(* Logix 5000 project; controller LeakTestAuto vendor 1 type 14 code 226 rev 37.11; software revision 37.01; part 3 of 14 *)

        [3].Detailed.element_data[8].Variable_code := 59, [3].Detailed.element_data[8].prec_code := 2, [3].Detailed.element_data[8].Unit_code := 60, [3].Detailed.element_data[8].result_measurement := 1.0002404, [3].Detailed.element_data[9].Variable_code := 12, [3].Detailed.element_data[9].prec_code := 3, [3].Detailed.element_data[9].Unit_code := 12, [3].Detailed.element_data[9].result_measurement := 5.000001, [3].Detailed.element_data[10].Variable_code := 62, [3].Detailed.element_data[10].prec_code := 2, [3].Detailed.element_data[10].Unit_code := 60, [3].Detailed.element_data[10].result_measurement := 1.1002644, [3].Detailed.element_data[11].Variable_code := 21, [3].Detailed.element_data[11].prec_code := 3, [3].Detailed.element_data[11].Unit_code := 41, [3].Detailed.element_data[11].result_measurement := 0.0015180558, [3].Detailed.element_data[12].Variable_code := 25, [3].Detailed.element_data[12].prec_code := 3, [3].Detailed.element_data[12].Unit_code := 41, [3].Detailed.element_data[12].result_measurement := 0.021727756, [3].Detailed.element_data[13].Variable_code := 216, [3].Detailed.element_data[13].prec_code := 3, [3].Detailed.element_data[13].Unit_code := 41, [3].Detailed.element_data[13].result_measurement := 0.00085681677, [3].Detailed.element_data[14].Variable_code := 218, [3].Detailed.element_data[14].prec_code := 3, [3].Detailed.element_data[14].Unit_code := 41, [3].Detailed.element_data[14].result_measurement := 0.01094304, [3].Detailed.element_data[15].Variable_code := 295, [3].Detailed.element_data[15].prec_code := 3, [3].Detailed.element_data[15].Unit_code := 12, [3].Detailed.element_data[15].result_measurement := 5.1383443, [4].UID := 41965, [4].Basic.unique_id := 41965, [4].Basic.channel_num := 1, [4].Basic.program_num := 2, [4].Basic.evaluation_code := 1, [4].Basic.test_port := 1, [4].Basic.year := 26, [4].Basic.month := 6, [4].Basic.date := 4, [4].Basic.hour := 15, [4].Basic.minute := 7, [4].Basic.second := 53, [4].Basic.flags := 12, [4].Basic.Num_tests := 1, [4].Basic.test_elements.test_type := 66, [4].Basic.test_elements.test_eval := 1, [4].Basic.test_elements.num_elements := 16, [4].Detailed.unique_id := 41965, [4].Detailed.num_elements := 16, [4].Detailed.Test_Type := 66, [4].Detailed.element_data[0].Variable_code := 61, [4].Detailed.element_data[0].prec_code := 2, [4].Detailed.element_data[0].Unit_code := 60, [4].Detailed.element_data[0].result_measurement := -0.06593764, [4].Detailed.element_data[1].Variable_code := 28, [4].Detailed.element_data[1].prec_code := 3, [4].Detailed.element_data[1].Unit_code := 41, [4].Detailed.element_data[1].result_measurement := 0.00029802322,
        [4].Detailed.element_data[2].Variable_code := 13, [4].Detailed.element_data[2].prec_code := 3, [4].Detailed.element_data[2].Unit_code := 12, [4].Detailed.element_data[2].result_measurement := 5.1366444, [4].Detailed.element_data[3].Variable_code := 75, [4].Detailed.element_data[3].prec_code := 2, [4].Detailed.element_data[3].Unit_code := 60, [4].Detailed.element_data[4].Variable_code := 60, [4].Detailed.element_data[4].prec_code := 2, [4].Detailed.element_data[4].Unit_code := 60, [4].Detailed.element_data[4].result_measurement := -0.06984919, [4].Detailed.element_data[5].Variable_code := 56, [4].Detailed.element_data[5].prec_code := 3, [4].Detailed.element_data[5].Unit_code := 41, [4].Detailed.element_data[5].result_measurement := 0.00021420419, [4].Detailed.element_data[6].Variable_code := 55, [4].Detailed.element_data[6].prec_code := 3, [4].Detailed.element_data[6].Unit_code := 12, [4].Detailed.element_data[6].result_measurement := 5.1366444, [4].Detailed.element_data[7].Variable_code := 58, [4].Detailed.element_data[7].prec_code := 2, [4].Detailed.element_data[7].Unit_code := 60, [4].Detailed.element_data[7].result_measurement := -1.0002404, [4].Detailed.element_data[8].Variable_code := 59, [4].Detailed.element_data[8].prec_code := 2, [4].Detailed.element_data[8].Unit_code := 60, [4].Detailed.element_data[8].result_measurement := 1.0002404, [4].Detailed.element_data[9].Variable_code := 12, [4].Detailed.element_data[9].prec_code := 3, [4].Detailed.element_data[9].Unit_code := 12, [4].Detailed.element_data[9].result_measurement := 5.000001, [4].Detailed.element_data[10].Variable_code := 62, [4].Detailed.element_data[10].prec_code := 2, [4].Detailed.element_data[10].Unit_code := 60, [4].Detailed.element_data[10].result_measurement := 1.1002644, [4].Detailed.element_data[11].Variable_code := 21, [4].Detailed.element_data[11].prec_code := 3, [4].Detailed.element_data[11].Unit_code := 41, [4].Detailed.element_data[11].result_measurement := 0.0015180558, [4].Detailed.element_data[12].Variable_code := 25, [4].Detailed.element_data[12].prec_code := 3, [4].Detailed.element_data[12].Unit_code := 41, [4].Detailed.element_data[12].result_measurement := 0.021727756, [4].Detailed.element_data[13].Variable_code := 216, [4].Detailed.element_data[13].prec_code := 3, [4].Detailed.element_data[13].Unit_code := 41, [4].Detailed.element_data[13].result_measurement := 0.00085681677, [4].Detailed.element_data[14].Variable_code := 218, [4].Detailed.element_data[14].prec_code := 3, [4].Detailed.element_data[14].Unit_code := 41, [4].Detailed.element_data[14].result_measurement := 0.01094304, [4].Detailed.element_data[15].Variable_code := 295, [4].Detailed.element_data[15].prec_code := 3, [4].Detailed.element_data[15].Unit_code := 12, [4].Detailed.element_data[15].result_measurement := 5.138372, [5].UID := 41968, [5].Basic.unique_id := 41968, [5].Basic.channel_num := 1, [5].Basic.program_num := 2, [5].Basic.evaluation_code := 1,
        [5].Basic.test_port := 1, [5].Basic.year := 26, [5].Basic.month := 6, [5].Basic.date := 4, [5].Basic.hour := 15, [5].Basic.minute := 9, [5].Basic.second := 31, [5].Basic.flags := 12, [5].Basic.Num_tests := 1, [5].Basic.test_elements.test_type := 66, [5].Basic.test_elements.test_eval := 1, [5].Basic.test_elements.num_elements := 16, [5].Detailed.unique_id := 41968, [5].Detailed.num_elements := 16, [5].Detailed.Test_Type := 66, [5].Detailed.element_data[0].Variable_code := 61, [5].Detailed.element_data[0].prec_code := 2, [5].Detailed.element_data[0].Unit_code := 60, [5].Detailed.element_data[0].result_measurement := -0.054761767, [5].Detailed.element_data[1].Variable_code := 28, [5].Detailed.element_data[1].prec_code := 3, [5].Detailed.element_data[1].Unit_code := 41, [5].Detailed.element_data[1].result_measurement := 0.0005075708, [5].Detailed.element_data[2].Variable_code := 13, [5].Detailed.element_data[2].prec_code := 3, [5].Detailed.element_data[2].Unit_code := 12, [5].Detailed.element_data[2].result_measurement := 5.1372128, [5].Detailed.element_data[3].Variable_code := 75, [5].Detailed.element_data[3].prec_code := 2, [5].Detailed.element_data[3].Unit_code := 60, [5].Detailed.element_data[4].Variable_code := 60, [5].Detailed.element_data[4].prec_code := 2, [5].Detailed.element_data[4].Unit_code := 60, [5].Detailed.element_data[4].result_measurement := -0.05811453, [5].Detailed.element_data[5].Variable_code := 56, [5].Detailed.element_data[5].prec_code := 3, [5].Detailed.element_data[5].Unit_code := 41, [5].Detailed.element_data[5].result_measurement := 0.0003213063, [5].Detailed.element_data[6].Variable_code := 55, [5].Detailed.element_data[6].prec_code := 3, [5].Detailed.element_data[6].Unit_code := 12, [5].Detailed.element_data[6].result_measurement := 5.1372128, [5].Detailed.element_data[7].Variable_code := 58, [5].Detailed.element_data[7].prec_code := 2, [5].Detailed.element_data[7].Unit_code := 60, [5].Detailed.element_data[7].result_measurement := -1.0002404, [5].Detailed.element_data[8].Variable_code := 59, [5].Detailed.element_data[8].prec_code := 2, [5].Detailed.element_data[8].Unit_code := 60, [5].Detailed.element_data[8].result_measurement := 1.0002404, [5].Detailed.element_data[9].Variable_code := 12, [5].Detailed.element_data[9].prec_code := 3, [5].Detailed.element_data[9].Unit_code := 12, [5].Detailed.element_data[9].result_measurement := 5.000001, [5].Detailed.element_data[10].Variable_code := 62, [5].Detailed.element_data[10].prec_code := 2, [5].Detailed.element_data[10].Unit_code := 60, [5].Detailed.element_data[10].result_measurement := 1.1002644, [5].Detailed.element_data[11].Variable_code := 21, [5].Detailed.element_data[11].prec_code := 3,
        [5].Detailed.element_data[11].Unit_code := 41, [5].Detailed.element_data[11].result_measurement := 0.0015180558, [5].Detailed.element_data[12].Variable_code := 25, [5].Detailed.element_data[12].prec_code := 3, [5].Detailed.element_data[12].Unit_code := 41, [5].Detailed.element_data[12].result_measurement := 0.021727756, [5].Detailed.element_data[13].Variable_code := 216, [5].Detailed.element_data[13].prec_code := 3, [5].Detailed.element_data[13].Unit_code := 41, [5].Detailed.element_data[13].result_measurement := 0.00085681677, [5].Detailed.element_data[14].Variable_code := 218, [5].Detailed.element_data[14].prec_code := 3, [5].Detailed.element_data[14].Unit_code := 41, [5].Detailed.element_data[14].result_measurement := 0.01094304, [5].Detailed.element_data[15].Variable_code := 295, [5].Detailed.element_data[15].prec_code := 3, [5].Detailed.element_data[15].Unit_code := 12, [5].Detailed.element_data[15].result_measurement := 5.139271, [6].UID := 42010, [6].Basic.unique_id := 42010, [6].Basic.channel_num := 1, [6].Basic.program_num := 2, [6].Basic.evaluation_code := 1, [6].Basic.test_port := 1, [6].Basic.year := 26, [6].Basic.month := 6, [6].Basic.date := 5, [6].Basic.hour := 10, [6].Basic.minute := 13, [6].Basic.second := 42, [6].Basic.flags := 12, [6].Basic.Num_tests := 1, [6].Basic.test_elements.test_type := 66, [6].Basic.test_elements.test_eval := 1, [6].Basic.test_elements.num_elements := 16, [6].Detailed.unique_id := 42010, [6].Detailed.num_elements := 16, [6].Detailed.Test_Type := 66, [6].Detailed.element_data[0].Variable_code := 61, [6].Detailed.element_data[0].prec_code := 2, [6].Detailed.element_data[0].Unit_code := 60, [6].Detailed.element_data[0].result_measurement := -0.067055225, [6].Detailed.element_data[1].Variable_code := 28, [6].Detailed.element_data[1].prec_code := 3, [6].Detailed.element_data[1].Unit_code := 41, [6].Detailed.element_data[1].result_measurement := 0.00027939677, [6].Detailed.element_data[2].Variable_code := 13, [6].Detailed.element_data[2].prec_code := 3, [6].Detailed.element_data[2].Unit_code := 12, [6].Detailed.element_data[2].result_measurement := 5.1023254, [6].Detailed.element_data[3].Variable_code := 75, [6].Detailed.element_data[3].prec_code := 2, [6].Detailed.element_data[3].Unit_code := 60, [6].Detailed.element_data[4].Variable_code := 60, [6].Detailed.element_data[4].prec_code := 2, [6].Detailed.element_data[4].Unit_code := 60, [6].Detailed.element_data[4].result_measurement := -0.07208437, [6].Detailed.element_data[5].Variable_code := 56, [6].Detailed.element_data[5].prec_code := 3, [6].Detailed.element_data[5].Unit_code := 41,
        [6].Detailed.element_data[5].result_measurement := 0.00019092113, [6].Detailed.element_data[6].Variable_code := 55, [6].Detailed.element_data[6].prec_code := 3, [6].Detailed.element_data[6].Unit_code := 12, [6].Detailed.element_data[6].result_measurement := 5.1023254, [6].Detailed.element_data[7].Variable_code := 58, [6].Detailed.element_data[7].prec_code := 2, [6].Detailed.element_data[7].Unit_code := 60, [6].Detailed.element_data[7].result_measurement := -1.0002404, [6].Detailed.element_data[8].Variable_code := 59, [6].Detailed.element_data[8].prec_code := 2, [6].Detailed.element_data[8].Unit_code := 60, [6].Detailed.element_data[8].result_measurement := 1.0002404, [6].Detailed.element_data[9].Variable_code := 12, [6].Detailed.element_data[9].prec_code := 3, [6].Detailed.element_data[9].Unit_code := 12, [6].Detailed.element_data[9].result_measurement := 5.000001, [6].Detailed.element_data[10].Variable_code := 62, [6].Detailed.element_data[10].prec_code := 2, [6].Detailed.element_data[10].Unit_code := 60, [6].Detailed.element_data[10].result_measurement := 1.1002644, [6].Detailed.element_data[11].Variable_code := 21, [6].Detailed.element_data[11].prec_code := 3, [6].Detailed.element_data[11].Unit_code := 41, [6].Detailed.element_data[11].result_measurement := 0.0015180558, [6].Detailed.element_data[12].Variable_code := 25, [6].Detailed.element_data[12].prec_code := 3, [6].Detailed.element_data[12].Unit_code := 41, [6].Detailed.element_data[12].result_measurement := 0.021727756, [6].Detailed.element_data[13].Variable_code := 216, [6].Detailed.element_data[13].prec_code := 3, [6].Detailed.element_data[13].Unit_code := 41, [6].Detailed.element_data[13].result_measurement := 0.00085681677, [6].Detailed.element_data[14].Variable_code := 218, [6].Detailed.element_data[14].prec_code := 3, [6].Detailed.element_data[14].Unit_code := 41, [6].Detailed.element_data[14].result_measurement := 0.01094304, [6].Detailed.element_data[15].Variable_code := 295, [6].Detailed.element_data[15].prec_code := 3, [6].Detailed.element_data[15].Unit_code := 12, [6].Detailed.element_data[15].result_measurement := 5.1039925, [7].UID := 42013, [7].Basic.unique_id := 42013, [7].Basic.channel_num := 1, [7].Basic.program_num := 2, [7].Basic.evaluation_code := 1, [7].Basic.test_port := 1, [7].Basic.year := 26, [7].Basic.month := 6, [7].Basic.date := 5, [7].Basic.hour := 10, [7].Basic.minute := 17, [7].Basic.second := 34, [7].Basic.flags := 12, [7].Basic.Num_tests := 1, [7].Basic.test_elements.test_type := 66, [7].Basic.test_elements.test_eval := 1, [7].Basic.test_elements.num_elements := 16, [7].Detailed.unique_id := 42013, [7].Detailed.num_elements := 16,
        [7].Detailed.Test_Type := 66, [7].Detailed.element_data[0].Variable_code := 61, [7].Detailed.element_data[0].prec_code := 2, [7].Detailed.element_data[0].Unit_code := 60, [7].Detailed.element_data[0].result_measurement := -0.07040799, [7].Detailed.element_data[1].Variable_code := 28, [7].Detailed.element_data[1].prec_code := 3, [7].Detailed.element_data[1].Unit_code := 41, [7].Detailed.element_data[1].result_measurement := 0.00022351742, [7].Detailed.element_data[2].Variable_code := 13, [7].Detailed.element_data[2].prec_code := 3, [7].Detailed.element_data[2].Unit_code := 12, [7].Detailed.element_data[2].result_measurement := 5.101585, [7].Detailed.element_data[3].Variable_code := 75, [7].Detailed.element_data[3].prec_code := 2, [7].Detailed.element_data[3].Unit_code := 60, [7].Detailed.element_data[4].Variable_code := 60, [7].Detailed.element_data[4].prec_code := 2, [7].Detailed.element_data[4].Unit_code := 60, [7].Detailed.element_data[4].result_measurement := -0.07711351, [7].Detailed.element_data[5].Variable_code := 56, [7].Detailed.element_data[5].prec_code := 3, [7].Detailed.element_data[5].Unit_code := 41, [7].Detailed.element_data[5].result_measurement := 0.00014901161, [7].Detailed.element_data[6].Variable_code := 55, [7].Detailed.element_data[6].prec_code := 3, [7].Detailed.element_data[6].Unit_code := 12, [7].Detailed.element_data[6].result_measurement := 5.101585, [7].Detailed.element_data[7].Variable_code := 58, [7].Detailed.element_data[7].prec_code := 2, [7].Detailed.element_data[7].Unit_code := 60, [7].Detailed.element_data[7].result_measurement := -1.0002404, [7].Detailed.element_data[8].Variable_code := 59, [7].Detailed.element_data[8].prec_code := 2, [7].Detailed.element_data[8].Unit_code := 60, [7].Detailed.element_data[8].result_measurement := 1.0002404, [7].Detailed.element_data[9].Variable_code := 12, [7].Detailed.element_data[9].prec_code := 3, [7].Detailed.element_data[9].Unit_code := 12, [7].Detailed.element_data[9].result_measurement := 5.000001, [7].Detailed.element_data[10].Variable_code := 62, [7].Detailed.element_data[10].prec_code := 2, [7].Detailed.element_data[10].Unit_code := 60, [7].Detailed.element_data[10].result_measurement := 1.1002644, [7].Detailed.element_data[11].Variable_code := 21, [7].Detailed.element_data[11].prec_code := 3, [7].Detailed.element_data[11].Unit_code := 41, [7].Detailed.element_data[11].result_measurement := 0.0015180558, [7].Detailed.element_data[12].Variable_code := 25, [7].Detailed.element_data[12].prec_code := 3, [7].Detailed.element_data[12].Unit_code := 41, [7].Detailed.element_data[12].result_measurement := 0.021727756, [7].Detailed.element_data[13].Variable_code := 216, [7].Detailed.element_data[13].prec_code := 3, [7].Detailed.element_data[13].Unit_code := 41, [7].Detailed.element_data[13].result_measurement := 0.00085681677, [7].Detailed.element_data[14].Variable_code := 218, [7].Detailed.element_data[14].prec_code := 3, [7].Detailed.element_data[14].Unit_code := 41, [7].Detailed.element_data[14].result_measurement := 0.01094304,
        [7].Detailed.element_data[15].Variable_code := 295, [7].Detailed.element_data[15].prec_code := 3, [7].Detailed.element_data[15].Unit_code := 12, [7].Detailed.element_data[15].result_measurement := 5.103038, [8].UID := 42016, [8].Basic.unique_id := 42016, [8].Basic.channel_num := 1, [8].Basic.program_num := 2, [8].Basic.evaluation_code := 1, [8].Basic.test_port := 1, [8].Basic.year := 26, [8].Basic.month := 6, [8].Basic.date := 5, [8].Basic.hour := 10, [8].Basic.minute := 18, [8].Basic.second := 33, [8].Basic.flags := 12, [8].Basic.Num_tests := 1, [8].Basic.test_elements.test_type := 66, [8].Basic.test_elements.test_eval := 1, [8].Basic.test_elements.num_elements := 16, [8].Detailed.unique_id := 42016, [8].Detailed.num_elements := 16, [8].Detailed.Test_Type := 66, [8].Detailed.element_data[0].Variable_code := 61, [8].Detailed.element_data[0].prec_code := 2, [8].Detailed.element_data[0].Unit_code := 60, [8].Detailed.element_data[0].result_measurement := -0.0692904, [8].Detailed.element_data[1].Variable_code := 28, [8].Detailed.element_data[1].prec_code := 3, [8].Detailed.element_data[1].Unit_code := 41, [8].Detailed.element_data[1].result_measurement := 0.00023748726, [8].Detailed.element_data[2].Variable_code := 13, [8].Detailed.element_data[2].prec_code := 3, [8].Detailed.element_data[2].Unit_code := 12, [8].Detailed.element_data[2].result_measurement := 5.1036057, [8].Detailed.element_data[3].Variable_code := 75, [8].Detailed.element_data[3].prec_code := 2, [8].Detailed.element_data[3].Unit_code := 60, [8].Detailed.element_data[4].Variable_code := 60, [8].Detailed.element_data[4].prec_code := 2, [8].Detailed.element_data[4].Unit_code := 60, [8].Detailed.element_data[4].result_measurement := -0.073201954, [8].Detailed.element_data[5].Variable_code := 56, [8].Detailed.element_data[5].prec_code := 3, [8].Detailed.element_data[5].Unit_code := 41, [8].Detailed.element_data[5].result_measurement := 0.0001816079, [8].Detailed.element_data[6].Variable_code := 55, [8].Detailed.element_data[6].prec_code := 3, [8].Detailed.element_data[6].Unit_code := 12, [8].Detailed.element_data[6].result_measurement := 5.1036057, [8].Detailed.element_data[7].Variable_code := 58, [8].Detailed.element_data[7].prec_code := 2, [8].Detailed.element_data[7].Unit_code := 60, [8].Detailed.element_data[7].result_measurement := -1.0002404, [8].Detailed.element_data[8].Variable_code := 59, [8].Detailed.element_data[8].prec_code := 2, [8].Detailed.element_data[8].Unit_code := 60, [8].Detailed.element_data[8].result_measurement := 1.0002404, [8].Detailed.element_data[9].Variable_code := 12,
        [8].Detailed.element_data[9].prec_code := 3, [8].Detailed.element_data[9].Unit_code := 12, [8].Detailed.element_data[9].result_measurement := 5.000001, [8].Detailed.element_data[10].Variable_code := 62, [8].Detailed.element_data[10].prec_code := 2, [8].Detailed.element_data[10].Unit_code := 60, [8].Detailed.element_data[10].result_measurement := 1.1002644, [8].Detailed.element_data[11].Variable_code := 21, [8].Detailed.element_data[11].prec_code := 3, [8].Detailed.element_data[11].Unit_code := 41, [8].Detailed.element_data[11].result_measurement := 0.0015180558, [8].Detailed.element_data[12].Variable_code := 25, [8].Detailed.element_data[12].prec_code := 3, [8].Detailed.element_data[12].Unit_code := 41, [8].Detailed.element_data[12].result_measurement := 0.021727756, [8].Detailed.element_data[13].Variable_code := 216, [8].Detailed.element_data[13].prec_code := 3, [8].Detailed.element_data[13].Unit_code := 41, [8].Detailed.element_data[13].result_measurement := 0.00085681677, [8].Detailed.element_data[14].Variable_code := 218, [8].Detailed.element_data[14].prec_code := 3, [8].Detailed.element_data[14].Unit_code := 41, [8].Detailed.element_data[14].result_measurement := 0.01094304, [8].Detailed.element_data[15].Variable_code := 295, [8].Detailed.element_data[15].prec_code := 3, [8].Detailed.element_data[15].Unit_code := 12, [8].Detailed.element_data[15].result_measurement := 5.1049933);
   CTS2_ResultHistoryVol : udt_CTS_RESULT[10] := ([0].UID := 41958, [0].Basic.unique_id := 41958, [0].Basic.channel_num := 1, [0].Basic.program_num := 1, [0].Basic.evaluation_code := 1, [0].Basic.test_port := 1, [0].Basic.year := 26, [0].Basic.month := 6, [0].Basic.date := 4, [0].Basic.hour := 15, [0].Basic.minute := 3, [0].Basic.second := 10, [0].Basic.flags := 12, [0].Basic.Num_tests := 1, [0].Basic.test_elements.test_type := 69, [0].Basic.test_elements.test_eval := 1, [0].Basic.test_elements.num_elements := 4, [0].Detailed.unique_id := 41958, [0].Detailed.num_elements := 4, [0].Detailed.Test_Type := 69, [0].Detailed.element_data[0].Variable_code := 245, [0].Detailed.element_data[0].prec_code := 2, [0].Detailed.element_data[0].Unit_code := 165, [0].Detailed.element_data[0].result_measurement := 186.90665, [0].Detailed.element_data[1].Variable_code := 13, [0].Detailed.element_data[1].prec_code := 3, [0].Detailed.element_data[1].Unit_code := 12, [0].Detailed.element_data[1].result_measurement := 1.7801206, [0].Detailed.element_data[2].Variable_code := 247, [0].Detailed.element_data[2].prec_code := 3, [0].Detailed.element_data[2].Unit_code := 12, [0].Detailed.element_data[2].result_measurement := 5.1072845, [0].Detailed.element_data[3].Variable_code := 295, [0].Detailed.element_data[3].prec_code := 3, [0].Detailed.element_data[3].Unit_code := 12, [0].Detailed.element_data[3].result_measurement := 5.1086583, [1].UID := 41961, [1].Basic.unique_id := 41961, [1].Basic.channel_num := 1, [1].Basic.program_num := 1, [1].Basic.evaluation_code := 1, [1].Basic.test_port := 1, [1].Basic.year := 26, [1].Basic.month := 6, [1].Basic.date := 4, [1].Basic.hour := 15, [1].Basic.minute := 6, [1].Basic.second := 33, [1].Basic.flags := 12, [1].Basic.Num_tests := 1, [1].Basic.test_elements.test_type := 69, [1].Basic.test_elements.test_eval := 1, [1].Basic.test_elements.num_elements := 4, [1].Detailed.unique_id := 41961, [1].Detailed.num_elements := 4, [1].Detailed.Test_Type := 69, [1].Detailed.element_data[0].Variable_code := 245, [1].Detailed.element_data[0].prec_code := 2, [1].Detailed.element_data[0].Unit_code := 165, [1].Detailed.element_data[0].result_measurement := 186.6259,
        [1].Detailed.element_data[1].Variable_code := 13, [1].Detailed.element_data[1].prec_code := 3, [1].Detailed.element_data[1].Unit_code := 12, [1].Detailed.element_data[1].result_measurement := 1.7820624, [1].Detailed.element_data[2].Variable_code := 247, [1].Detailed.element_data[2].prec_code := 3, [1].Detailed.element_data[2].Unit_code := 12, [1].Detailed.element_data[2].result_measurement := 5.1078525, [1].Detailed.element_data[3].Variable_code := 295, [1].Detailed.element_data[3].prec_code := 3, [1].Detailed.element_data[3].Unit_code := 12, [1].Detailed.element_data[3].result_measurement := 5.1083417, [2].UID := 41964, [2].Basic.unique_id := 41964, [2].Basic.channel_num := 1, [2].Basic.program_num := 1, [2].Basic.evaluation_code := 1, [2].Basic.test_port := 1, [2].Basic.year := 26, [2].Basic.month := 6, [2].Basic.date := 4, [2].Basic.hour := 15, [2].Basic.minute := 7, [2].Basic.second := 46, [2].Basic.flags := 12, [2].Basic.Num_tests := 1, [2].Basic.test_elements.test_type := 69, [2].Basic.test_elements.test_eval := 1, [2].Basic.test_elements.num_elements := 4, [2].Detailed.unique_id := 41964, [2].Detailed.num_elements := 4, [2].Detailed.Test_Type := 69, [2].Detailed.element_data[0].Variable_code := 245, [2].Detailed.element_data[0].prec_code := 2, [2].Detailed.element_data[0].Unit_code := 165, [2].Detailed.element_data[0].result_measurement := 186.70047, [2].Detailed.element_data[1].Variable_code := 13, [2].Detailed.element_data[1].prec_code := 3, [2].Detailed.element_data[1].Unit_code := 12, [2].Detailed.element_data[1].result_measurement := 1.7814804, [2].Detailed.element_data[2].Variable_code := 247, [2].Detailed.element_data[2].prec_code := 3, [2].Detailed.element_data[2].Unit_code := 12, [2].Detailed.element_data[2].result_measurement := 5.1075125, [2].Detailed.element_data[3].Variable_code := 295, [2].Detailed.element_data[3].prec_code := 3, [2].Detailed.element_data[3].Unit_code := 12, [2].Detailed.element_data[3].result_measurement := 5.1079783, [3].UID := 41967, [3].Basic.unique_id := 41967, [3].Basic.channel_num := 1, [3].Basic.program_num := 1, [3].Basic.evaluation_code := 1, [3].Basic.test_port := 1, [3].Basic.year := 26, [3].Basic.month := 6, [3].Basic.date := 4, [3].Basic.hour := 15, [3].Basic.minute := 9, [3].Basic.second := 24,
        [3].Basic.flags := 12, [3].Basic.Num_tests := 1, [3].Basic.test_elements.test_type := 69, [3].Basic.test_elements.test_eval := 1, [3].Basic.test_elements.num_elements := 4, [3].Detailed.unique_id := 41967, [3].Detailed.num_elements := 4, [3].Detailed.Test_Type := 69, [3].Detailed.element_data[0].Variable_code := 245, [3].Detailed.element_data[0].prec_code := 2, [3].Detailed.element_data[0].Unit_code := 165, [3].Detailed.element_data[0].result_measurement := 186.79054, [3].Detailed.element_data[1].Variable_code := 13, [3].Detailed.element_data[1].prec_code := 3, [3].Detailed.element_data[1].Unit_code := 12, [3].Detailed.element_data[1].result_measurement := 1.7802324, [3].Detailed.element_data[2].Variable_code := 247, [3].Detailed.element_data[2].prec_code := 3, [3].Detailed.element_data[2].Unit_code := 12, [3].Detailed.element_data[2].result_measurement := 5.1055384, [3].Detailed.element_data[3].Variable_code := 295, [3].Detailed.element_data[3].prec_code := 3, [3].Detailed.element_data[3].Unit_code := 12, [3].Detailed.element_data[3].result_measurement := 5.1066375, [4].UID := 42009, [4].Basic.unique_id := 42009, [4].Basic.channel_num := 1, [4].Basic.program_num := 1, [4].Basic.evaluation_code := 1, [4].Basic.test_port := 1, [4].Basic.year := 26, [4].Basic.month := 6, [4].Basic.date := 5, [4].Basic.hour := 10, [4].Basic.minute := 13, [4].Basic.second := 35, [4].Basic.flags := 12, [4].Basic.Num_tests := 1, [4].Basic.test_elements.test_type := 69, [4].Basic.test_elements.test_eval := 1, [4].Basic.test_elements.num_elements := 4, [4].Detailed.unique_id := 42009, [4].Detailed.num_elements := 4, [4].Detailed.Test_Type := 69, [4].Detailed.element_data[0].Variable_code := 245, [4].Detailed.element_data[0].prec_code := 2, [4].Detailed.element_data[0].Unit_code := 165, [4].Detailed.element_data[0].result_measurement := 185.74803, [4].Detailed.element_data[1].Variable_code := 13, [4].Detailed.element_data[1].prec_code := 3, [4].Detailed.element_data[1].Unit_code := 12, [4].Detailed.element_data[1].result_measurement := 1.7781556, [4].Detailed.element_data[2].Variable_code := 247, [4].Detailed.element_data[2].prec_code := 3, [4].Detailed.element_data[2].Unit_code := 12, [4].Detailed.element_data[2].result_measurement := 5.0810447, [4].Detailed.element_data[3].Variable_code := 295, [4].Detailed.element_data[3].prec_code := 3, [4].Detailed.element_data[3].Unit_code := 12, [4].Detailed.element_data[3].result_measurement := 5.081105,
        [5].UID := 42012, [5].Basic.unique_id := 42012, [5].Basic.channel_num := 1, [5].Basic.program_num := 1, [5].Basic.evaluation_code := 1, [5].Basic.test_port := 1, [5].Basic.year := 26, [5].Basic.month := 6, [5].Basic.date := 5, [5].Basic.hour := 10, [5].Basic.minute := 17, [5].Basic.second := 27, [5].Basic.flags := 12, [5].Basic.Num_tests := 1, [5].Basic.test_elements.test_type := 69, [5].Basic.test_elements.test_eval := 1, [5].Basic.test_elements.num_elements := 4, [5].Detailed.unique_id := 42012, [5].Detailed.num_elements := 4, [5].Detailed.Test_Type := 69, [5].Detailed.element_data[0].Variable_code := 245, [5].Detailed.element_data[0].prec_code := 2, [5].Detailed.element_data[0].Unit_code := 165, [5].Detailed.element_data[0].result_measurement := 185.72876, [5].Detailed.element_data[1].Variable_code := 13, [5].Detailed.element_data[1].prec_code := 3, [5].Detailed.element_data[1].Unit_code := 12, [5].Detailed.element_data[1].result_measurement := 1.7785281, [5].Detailed.element_data[2].Variable_code := 247, [5].Detailed.element_data[2].prec_code := 3, [5].Detailed.element_data[2].Unit_code := 12, [5].Detailed.element_data[2].result_measurement := 5.081766, [5].Detailed.element_data[3].Variable_code := 295, [5].Detailed.element_data[3].prec_code := 3, [5].Detailed.element_data[3].Unit_code := 12, [5].Detailed.element_data[3].result_measurement := 5.0830374, [6].UID := 42015, [6].Basic.unique_id := 42015, [6].Basic.channel_num := 1, [6].Basic.program_num := 1, [6].Basic.evaluation_code := 1, [6].Basic.test_port := 1, [6].Basic.year := 26, [6].Basic.month := 6, [6].Basic.date := 5, [6].Basic.hour := 10, [6].Basic.minute := 18, [6].Basic.second := 26, [6].Basic.flags := 12, [6].Basic.Num_tests := 1, [6].Basic.test_elements.test_type := 69, [6].Basic.test_elements.test_eval := 1, [6].Basic.test_elements.num_elements := 4, [6].Detailed.unique_id := 42015, [6].Detailed.num_elements := 4, [6].Detailed.Test_Type := 69, [6].Detailed.element_data[0].Variable_code := 245, [6].Detailed.element_data[0].prec_code := 2, [6].Detailed.element_data[0].Unit_code := 165, [6].Detailed.element_data[0].result_measurement := 185.95625,
        [6].Detailed.element_data[1].Variable_code := 13, [6].Detailed.element_data[1].prec_code := 3, [6].Detailed.element_data[1].Unit_code := 12, [6].Detailed.element_data[1].result_measurement := 1.778258, [6].Detailed.element_data[2].Variable_code := 247, [6].Detailed.element_data[2].prec_code := 3, [6].Detailed.element_data[2].Unit_code := 12, [6].Detailed.element_data[2].result_measurement := 5.08504, [6].Detailed.element_data[3].Variable_code := 295, [6].Detailed.element_data[3].prec_code := 3, [6].Detailed.element_data[3].Unit_code := 12, [6].Detailed.element_data[3].result_measurement := 5.086218, [7].UID := 42018, [7].Basic.unique_id := 42018, [7].Basic.channel_num := 1, [7].Basic.program_num := 1, [7].Basic.evaluation_code := 2, [7].Basic.test_port := 1, [7].Basic.year := 26, [7].Basic.month := 6, [7].Basic.date := 5, [7].Basic.hour := 10, [7].Basic.minute := 54, [7].Basic.second := 14, [7].Basic.flags := 12, [7].Basic.Num_tests := 1, [7].Basic.test_elements.test_type := 69, [7].Basic.test_elements.test_eval := 2, [7].Basic.test_elements.num_elements := 4, [7].Detailed.unique_id := 42018, [7].Detailed.num_elements := 4, [7].Detailed.Test_Type := 69, [7].Detailed.element_data[0].Variable_code := 245, [7].Detailed.element_data[0].prec_code := 2, [7].Detailed.element_data[0].Unit_code := 165, [7].Detailed.element_data[0].result_measurement := 1000.0, [7].Detailed.element_data[1].Variable_code := 13, [7].Detailed.element_data[1].prec_code := 3, [7].Detailed.element_data[1].Unit_code := 12, [7].Detailed.element_data[1].result_measurement := 0.0002933666, [7].Detailed.element_data[2].Variable_code := 247, [7].Detailed.element_data[2].prec_code := 3, [7].Detailed.element_data[2].Unit_code := 12, [7].Detailed.element_data[2].result_measurement := 5.0650864, [7].Detailed.element_data[3].Variable_code := 295, [7].Detailed.element_data[3].prec_code := 3, [7].Detailed.element_data[3].Unit_code := 12, [7].Detailed.element_data[3].result_measurement := 5.0667486, [8].UID := 42020, [8].Basic.unique_id := 42020, [8].Basic.channel_num := 1, [8].Basic.program_num := 1, [8].Basic.evaluation_code := 1, [8].Basic.test_port := 1, [8].Basic.year := 26, [8].Basic.month := 6, [8].Basic.date := 5, [8].Basic.hour := 10, [8].Basic.minute := 54, [8].Basic.second := 35,
        [8].Basic.flags := 12, [8].Basic.Num_tests := 1, [8].Basic.test_elements.test_type := 69, [8].Basic.test_elements.test_eval := 1, [8].Basic.test_elements.num_elements := 4, [8].Detailed.unique_id := 42020, [8].Detailed.num_elements := 4, [8].Detailed.Test_Type := 69, [8].Detailed.element_data[0].Variable_code := 245, [8].Detailed.element_data[0].prec_code := 2, [8].Detailed.element_data[0].Unit_code := 165, [8].Detailed.element_data[0].result_measurement := 186.5566, [8].Detailed.element_data[1].Variable_code := 13, [8].Detailed.element_data[1].prec_code := 3, [8].Detailed.element_data[1].Unit_code := 12, [8].Detailed.element_data[1].result_measurement := 1.768372, [8].Detailed.element_data[2].Variable_code := 247, [8].Detailed.element_data[2].prec_code := 3, [8].Detailed.element_data[2].Unit_code := 12, [8].Detailed.element_data[2].result_measurement := 5.0673866, [8].Detailed.element_data[3].Variable_code := 295, [8].Detailed.element_data[3].prec_code := 3, [8].Detailed.element_data[3].Unit_code := 12, [8].Detailed.element_data[3].result_measurement := 5.068574, [9].UID := 42023, [9].Basic.unique_id := 42023, [9].Basic.channel_num := 1, [9].Basic.program_num := 1, [9].Basic.evaluation_code := 1, [9].Basic.test_port := 1, [9].Basic.year := 26, [9].Basic.month := 6, [9].Basic.date := 5, [9].Basic.hour := 10, [9].Basic.minute := 55, [9].Basic.second := 43, [9].Basic.flags := 12, [9].Basic.Num_tests := 1, [9].Basic.test_elements.test_type := 69, [9].Basic.test_elements.test_eval := 1, [9].Basic.test_elements.num_elements := 4, [9].Detailed.unique_id := 42023, [9].Detailed.num_elements := 4, [9].Detailed.Test_Type := 69, [9].Detailed.element_data[0].Variable_code := 245, [9].Detailed.element_data[0].prec_code := 2, [9].Detailed.element_data[0].Unit_code := 165, [9].Detailed.element_data[0].result_measurement := 186.64526, [9].Detailed.element_data[1].Variable_code := 13, [9].Detailed.element_data[1].prec_code := 3, [9].Detailed.element_data[1].Unit_code := 12, [9].Detailed.element_data[1].result_measurement := 1.7689215, [9].Detailed.element_data[2].Variable_code := 247, [9].Detailed.element_data[2].prec_code := 3, [9].Detailed.element_data[2].Unit_code := 12, [9].Detailed.element_data[2].result_measurement := 5.07053, [9].Detailed.element_data[3].Variable_code := 295, [9].Detailed.element_data[3].prec_code := 3, [9].Detailed.element_data[3].Unit_code := 12, [9].Detailed.element_data[3].result_measurement := 5.0715685);
   CTS2_Seq : udt_SequenceStructure_X64 := (CycleDone := 1, CurrentStep := 9000, NextStep := 9000, ONS := -32767, StepHistory[0] := 1000, StepHistory[1] := 1010, StepHistory[2] := 1020, StepHistory[3] := 1030, StepHistory[4] := 2000, StepHistory[5] := 2010, StepHistory[6] := 2020, StepHistory[7] := 2030, StepHistory[8] := 2000, StepHistory[9] := 2010, StepHistory[10] := 2020, StepHistory[11] := 2030, StepHistory[12] := 9000, StepHistory[13] := 1000, StepHistory[14] := 1010, StepHistory[15] := 1020, StepHistory[16] := 1030, StepHistory[17] := 2000, StepHistory[18] := 2010, StepHistory[19] := 2020, StepHistory[20] := 2030, StepHistory[21] := 2000, StepHistory[22] := 2010, StepHistory[23] := 2020, StepHistory[24] := 2030, StepHistory[25] := 9000, StepHistory[26] := 1000, StepHistory[27] := 1010, StepHistory[28] := 1020, StepHistory[29] := 1030, StepHistory[30] := 2000, StepHistory[31] := 2010, StepHistory[32] := 2020, StepHistory[33] := 2030, StepHistory[34] := 9000, StepHistory[35] := 1000, StepHistory[36] := 1010, StepHistory[37] := 1020, StepHistory[38] := 1030, StepHistory[39] := 2000, StepHistory[40] := 2010, StepHistory[41] := 2020, StepHistory[42] := 2030, StepHistory[43] := 2000, StepHistory[44] := 2010, StepHistory[45] := 2020, StepHistory[46] := 2030, StepHistory[47] := 9000, StepHistory[48] := 1000, StepHistory[49] := 1010, StepHistory[50] := 1020, StepHistory[51] := 1030, StepHistory[52] := 2000, StepHistory[53] := 2010, StepHistory[54] := 2020, StepHistory[55] := 2030,
        StepHistory[56] := 2000, StepHistory[57] := 2010, StepHistory[58] := 2020, StepHistory[59] := 2030, StepHistory[60] := 9000, StepHistory[61] := 1000, StepHistory[62] := 1010, StepHistory[63] := 1020, AverageCycleTime := 1.0542, CycleTimeHistory[0] := 2.209, CycleTimeHistory[1] := 2.209, CycleTimeHistory[3] := 1.206, CycleTimeHistory[4] := 2.209, CycleTimeHistory[5] := 2.209, CycleTimeHistory[8] := 0.5, StepTimeHistory[1] := 0.199, StepTimeHistory[2] := 0.199, StepTimeHistory[3] := 0.199, StepTimeHistory[5] := 1.0, StepTimeHistory[6] := 1.0, StepTimeHistory[7] := 1.0, StepTimeHistory[9] := 0.999, StepTimeHistory[10] := 0.999, StepTimeHistory[11] := 0.999, StepTimeHistory[12] := 0.999, StepTimeHistory[14] := 0.199, StepTimeHistory[15] := 0.199, StepTimeHistory[16] := 0.199, StepTimeHistory[18] := 1.0, StepTimeHistory[19] := 1.0, StepTimeHistory[20] := 1.0, StepTimeHistory[22] := 0.999, StepTimeHistory[23] := 0.999, StepTimeHistory[24] := 0.999, StepTimeHistory[27] := 0.199, StepTimeHistory[28] := 0.199, StepTimeHistory[29] := 0.199, StepTimeHistory[31] := 1.0, StepTimeHistory[32] := 1.0, StepTimeHistory[33] := 1.0, StepTimeHistory[34] := 1.0, StepTimeHistory[36] := 0.199, StepTimeHistory[37] := 0.199, StepTimeHistory[38] := 0.199, StepTimeHistory[40] := 0.999, StepTimeHistory[41] := 0.999, StepTimeHistory[42] := 0.999, StepTimeHistory[44] := 1.0, StepTimeHistory[45] := 1.0, StepTimeHistory[46] := 1.0, StepTimeHistory[47] := 1.0, StepTimeHistory[49] := 0.2, StepTimeHistory[50] := 0.2, StepTimeHistory[51] := 0.2, StepTimeHistory[53] := 0.999, StepTimeHistory[54] := 0.999, StepTimeHistory[55] := 0.999, StepTimeHistory[57] := 0.999, StepTimeHistory[58] := 0.999, StepTimeHistory[59] := 0.999,
        StepTimeHistory[62] := 0.199, StepTimeHistory[63] := 0.299, StepTimer.PRE := 999999999, CycleTimer.PRE := 999999999);
   CTS2_SeqUID : DINT := 42054;
   CTS2_UIDMsg : MESSAGE;
        MessageParameters(ServiceCode := 16#0010, LocalElement := CTS2_Result.UID, ...)
   CTS2_WriteMsg : MESSAGE;
        MessageParameters(ServiceCode := 16#0010, LocalElement := CTS2_BarcodeWrite.DATA[0], ...)
   CTS_NoResult : udt_CTS_RESULT;
   CTS_ResultDump : udt_CTS_RESULT := (UID := 41955, Basic.unique_id := 41955, Basic.channel_num := 1, Basic.program_num := 1, Basic.evaluation_code := 1, Basic.test_port := 1, Basic.year := 26, Basic.month := 6, Basic.date := 4, Basic.hour := 14, Basic.minute := 58, Basic.second := 18, Basic.flags := 12, Basic.Num_tests := 1, Basic.test_elements.test_type := 69, Basic.test_elements.test_eval := 1, Basic.test_elements.num_elements := 4, Detailed.unique_id := 41955, Detailed.num_elements := 4, Detailed.Test_Type := 69, Detailed.element_data[0].Variable_code := 245, Detailed.element_data[0].prec_code := 2, Detailed.element_data[0].Unit_code := 165, Detailed.element_data[0].result_measurement := 186.52744, Detailed.element_data[1].Variable_code := 13, Detailed.element_data[1].prec_code := 3, Detailed.element_data[1].Unit_code := 12, Detailed.element_data[1].result_measurement := 1.782449, Detailed.element_data[2].Variable_code := 247, Detailed.element_data[2].prec_code := 3, Detailed.element_data[2].Unit_code := 12, Detailed.element_data[2].result_measurement := 5.1072054, Detailed.element_data[3].Variable_code := 295, Detailed.element_data[3].prec_code := 3, Detailed.element_data[3].Unit_code := 12, Detailed.element_data[3].result_measurement := 5.109105);
   CurrentDUTData : udt_DUTHistory[2] := ([0].Barcode := 'B252620969', [0].VolumeTest.UID := 43022, [0].VolumeTest.Basic.unique_id := 43022, [0].VolumeTest.Basic.channel_num := 1, [0].VolumeTest.Basic.program_num := 1, [0].VolumeTest.Basic.evaluation_code := 2, [0].VolumeTest.Basic.test_port := 1, [0].VolumeTest.Basic.year := 26, [0].VolumeTest.Basic.month := 6, [0].VolumeTest.Basic.date := 5, [0].VolumeTest.Basic.hour := 10, [0].VolumeTest.Basic.minute := 56, [0].VolumeTest.Basic.second := 7, [0].VolumeTest.Basic.flags := 12, [0].VolumeTest.Basic.Num_tests := 1, [0].VolumeTest.Basic.test_elements.test_type := 69, [0].VolumeTest.Basic.test_elements.test_eval := 2, [0].VolumeTest.Basic.test_elements.num_elements := 4, [0].VolumeTest.Detailed.unique_id := 43022, [0].VolumeTest.Detailed.num_elements := 4, [0].VolumeTest.Detailed.Test_Type := 69, [0].VolumeTest.Detailed.element_data[0].Variable_code := 245, [0].VolumeTest.Detailed.element_data[0].prec_code := 2, [0].VolumeTest.Detailed.element_data[0].Unit_code := 165, [0].VolumeTest.Detailed.element_data[0].result_measurement := 1000.0, [0].VolumeTest.Detailed.element_data[1].Variable_code := 13, [0].VolumeTest.Detailed.element_data[1].prec_code := 3, [0].VolumeTest.Detailed.element_data[1].Unit_code := 12, [0].VolumeTest.Detailed.element_data[1].result_measurement := 0.0047218055, [0].VolumeTest.Detailed.element_data[2].Variable_code := 247, [0].VolumeTest.Detailed.element_data[2].prec_code := 3, [0].VolumeTest.Detailed.element_data[2].Unit_code := 12, [0].VolumeTest.Detailed.element_data[2].result_measurement := 5.095699, [0].VolumeTest.Detailed.element_data[3].Variable_code := 295, [0].VolumeTest.Detailed.element_data[3].prec_code := 3, [0].VolumeTest.Detailed.element_data[3].Unit_code := 12, [0].VolumeTest.Detailed.element_data[3].result_measurement := 5.096928, [0].LeakTest.UID := 43014, [0].LeakTest.Basic.unique_id := 43014, [0].LeakTest.Basic.channel_num := 1, [0].LeakTest.Basic.program_num := 2, [0].LeakTest.Basic.evaluation_code := 1, [0].LeakTest.Basic.test_port := 1, [0].LeakTest.Basic.year := 26, [0].LeakTest.Basic.month := 6, [0].LeakTest.Basic.date := 5, [0].LeakTest.Basic.hour := 10, [0].LeakTest.Basic.minute := 19, [0].LeakTest.Basic.second := 51, [0].LeakTest.Basic.flags := 12, [0].LeakTest.Basic.Num_tests := 1, [0].LeakTest.Basic.test_elements.test_type := 66, [0].LeakTest.Basic.test_elements.test_eval := 1, [0].LeakTest.Basic.test_elements.num_elements := 16, [0].LeakTest.Detailed.unique_id := 43014, [0].LeakTest.Detailed.num_elements := 16, [0].LeakTest.Detailed.Test_Type := 66, [0].LeakTest.Detailed.element_data[0].Variable_code := 61, [0].LeakTest.Detailed.element_data[0].prec_code := 2, [0].LeakTest.Detailed.element_data[0].Unit_code := 60,
        [0].LeakTest.Detailed.element_data[0].result_measurement := 0.007264316, [0].LeakTest.Detailed.element_data[1].Variable_code := 28, [0].LeakTest.Detailed.element_data[1].prec_code := 3, [0].LeakTest.Detailed.element_data[1].Unit_code := 41, [0].LeakTest.Detailed.element_data[1].result_measurement := 0.00015832484, [0].LeakTest.Detailed.element_data[2].Variable_code := 13, [0].LeakTest.Detailed.element_data[2].prec_code := 3, [0].LeakTest.Detailed.element_data[2].Unit_code := 12, [0].LeakTest.Detailed.element_data[2].result_measurement := 5.146228, [0].LeakTest.Detailed.element_data[3].Variable_code := 75, [0].LeakTest.Detailed.element_data[3].prec_code := 2, [0].LeakTest.Detailed.element_data[3].Unit_code := 60, [0].LeakTest.Detailed.element_data[4].Variable_code := 60, [0].LeakTest.Detailed.element_data[4].prec_code := 2, [0].LeakTest.Detailed.element_data[4].Unit_code := 60, [0].LeakTest.Detailed.element_data[4].result_measurement := 0.014528632, [0].LeakTest.Detailed.element_data[5].Variable_code := 56, [0].LeakTest.Detailed.element_data[5].prec_code := 3, [0].LeakTest.Detailed.element_data[5].Unit_code := 41, [0].LeakTest.Detailed.element_data[5].result_measurement := 0.00011641532, [0].LeakTest.Detailed.element_data[6].Variable_code := 55, [0].LeakTest.Detailed.element_data[6].prec_code := 3, [0].LeakTest.Detailed.element_data[6].Unit_code := 12, [0].LeakTest.Detailed.element_data[6].result_measurement := 5.146228, [0].LeakTest.Detailed.element_data[7].Variable_code := 58, [0].LeakTest.Detailed.element_data[7].prec_code := 2, [0].LeakTest.Detailed.element_data[7].Unit_code := 60, [0].LeakTest.Detailed.element_data[7].result_measurement := -1.0002404, [0].LeakTest.Detailed.element_data[8].Variable_code := 59, [0].LeakTest.Detailed.element_data[8].prec_code := 2, [0].LeakTest.Detailed.element_data[8].Unit_code := 60, [0].LeakTest.Detailed.element_data[8].result_measurement := 1.0002404, [0].LeakTest.Detailed.element_data[9].Variable_code := 12, [0].LeakTest.Detailed.element_data[9].prec_code := 3, [0].LeakTest.Detailed.element_data[9].Unit_code := 12, [0].LeakTest.Detailed.element_data[9].result_measurement := 5.000001, [0].LeakTest.Detailed.element_data[10].Variable_code := 62, [0].LeakTest.Detailed.element_data[10].prec_code := 2, [0].LeakTest.Detailed.element_data[10].Unit_code := 60, [0].LeakTest.Detailed.element_data[10].result_measurement := 1.1298805, [0].LeakTest.Detailed.element_data[11].Variable_code := 21, [0].LeakTest.Detailed.element_data[11].prec_code := 3, [0].LeakTest.Detailed.element_data[11].Unit_code := 41, [0].LeakTest.Detailed.element_data[11].result_measurement := 4.656613e-06, [0].LeakTest.Detailed.element_data[12].Variable_code := 25, [0].LeakTest.Detailed.element_data[12].prec_code := 3, [0].LeakTest.Detailed.element_data[12].Unit_code := 41, [0].LeakTest.Detailed.element_data[12].result_measurement := 0.023245811, [0].LeakTest.Detailed.element_data[13].Variable_code := 216, [0].LeakTest.Detailed.element_data[13].prec_code := 3, [0].LeakTest.Detailed.element_data[13].Unit_code := 41, [0].LeakTest.Detailed.element_data[13].result_measurement := -3.7252903e-05, [0].LeakTest.Detailed.element_data[14].Variable_code := 218, [0].LeakTest.Detailed.element_data[14].prec_code := 3, [0].LeakTest.Detailed.element_data[14].Unit_code := 41, [0].LeakTest.Detailed.element_data[14].result_measurement := 0.011632219, [0].LeakTest.Detailed.element_data[15].Variable_code := 295, [0].LeakTest.Detailed.element_data[15].prec_code := 3, [0].LeakTest.Detailed.element_data[15].Unit_code := 12, [0].LeakTest.Detailed.element_data[15].result_measurement := 5.14742,
        [1].Barcode := 'B252620970', [1].VolumeTest.UID := 42023, [1].VolumeTest.Basic.unique_id := 42023, [1].VolumeTest.Basic.channel_num := 1, [1].VolumeTest.Basic.program_num := 1, [1].VolumeTest.Basic.evaluation_code := 1, [1].VolumeTest.Basic.test_port := 1, [1].VolumeTest.Basic.year := 26, [1].VolumeTest.Basic.month := 6, [1].VolumeTest.Basic.date := 5, [1].VolumeTest.Basic.hour := 10, [1].VolumeTest.Basic.minute := 55, [1].VolumeTest.Basic.second := 43, [1].VolumeTest.Basic.flags := 12, [1].VolumeTest.Basic.Num_tests := 1, [1].VolumeTest.Basic.test_elements.test_type := 69, [1].VolumeTest.Basic.test_elements.test_eval := 1, [1].VolumeTest.Basic.test_elements.num_elements := 4, [1].VolumeTest.Detailed.unique_id := 42023, [1].VolumeTest.Detailed.num_elements := 4, [1].VolumeTest.Detailed.Test_Type := 69, [1].VolumeTest.Detailed.element_data[0].Variable_code := 245, [1].VolumeTest.Detailed.element_data[0].prec_code := 2, [1].VolumeTest.Detailed.element_data[0].Unit_code := 165, [1].VolumeTest.Detailed.element_data[0].result_measurement := 186.64526, [1].VolumeTest.Detailed.element_data[1].Variable_code := 13, [1].VolumeTest.Detailed.element_data[1].prec_code := 3, [1].VolumeTest.Detailed.element_data[1].Unit_code := 12, [1].VolumeTest.Detailed.element_data[1].result_measurement := 1.7689215, [1].VolumeTest.Detailed.element_data[2].Variable_code := 247, [1].VolumeTest.Detailed.element_data[2].prec_code := 3, [1].VolumeTest.Detailed.element_data[2].Unit_code := 12, [1].VolumeTest.Detailed.element_data[2].result_measurement := 5.07053, [1].VolumeTest.Detailed.element_data[3].Variable_code := 295, [1].VolumeTest.Detailed.element_data[3].prec_code := 3, [1].VolumeTest.Detailed.element_data[3].Unit_code := 12, [1].VolumeTest.Detailed.element_data[3].result_measurement := 5.0715685, [1].LeakTest.UID := 42016, [1].LeakTest.Basic.unique_id := 42016, [1].LeakTest.Basic.channel_num := 1, [1].LeakTest.Basic.program_num := 2, [1].LeakTest.Basic.evaluation_code := 1, [1].LeakTest.Basic.test_port := 1, [1].LeakTest.Basic.year := 26, [1].LeakTest.Basic.month := 6, [1].LeakTest.Basic.date := 5, [1].LeakTest.Basic.hour := 10, [1].LeakTest.Basic.minute := 18, [1].LeakTest.Basic.second := 33, [1].LeakTest.Basic.flags := 12, [1].LeakTest.Basic.Num_tests := 1, [1].LeakTest.Basic.test_elements.test_type := 66, [1].LeakTest.Basic.test_elements.test_eval := 1, [1].LeakTest.Basic.test_elements.num_elements := 16, [1].LeakTest.Detailed.unique_id := 42016, [1].LeakTest.Detailed.num_elements := 16, [1].LeakTest.Detailed.Test_Type := 66, [1].LeakTest.Detailed.element_data[0].Variable_code := 61, [1].LeakTest.Detailed.element_data[0].prec_code := 2, [1].LeakTest.Detailed.element_data[0].Unit_code := 60,
        [1].LeakTest.Detailed.element_data[0].result_measurement := -0.0692904, [1].LeakTest.Detailed.element_data[1].Variable_code := 28, [1].LeakTest.Detailed.element_data[1].prec_code := 3, [1].LeakTest.Detailed.element_data[1].Unit_code := 41, [1].LeakTest.Detailed.element_data[1].result_measurement := 0.00023748726, [1].LeakTest.Detailed.element_data[2].Variable_code := 13, [1].LeakTest.Detailed.element_data[2].prec_code := 3, [1].LeakTest.Detailed.element_data[2].Unit_code := 12, [1].LeakTest.Detailed.element_data[2].result_measurement := 5.1036057, [1].LeakTest.Detailed.element_data[3].Variable_code := 75, [1].LeakTest.Detailed.element_data[3].prec_code := 2, [1].LeakTest.Detailed.element_data[3].Unit_code := 60, [1].LeakTest.Detailed.element_data[4].Variable_code := 60, [1].LeakTest.Detailed.element_data[4].prec_code := 2, [1].LeakTest.Detailed.element_data[4].Unit_code := 60, [1].LeakTest.Detailed.element_data[4].result_measurement := -0.073201954, [1].LeakTest.Detailed.element_data[5].Variable_code := 56, [1].LeakTest.Detailed.element_data[5].prec_code := 3, [1].LeakTest.Detailed.element_data[5].Unit_code := 41, [1].LeakTest.Detailed.element_data[5].result_measurement := 0.0001816079, [1].LeakTest.Detailed.element_data[6].Variable_code := 55, [1].LeakTest.Detailed.element_data[6].prec_code := 3, [1].LeakTest.Detailed.element_data[6].Unit_code := 12, [1].LeakTest.Detailed.element_data[6].result_measurement := 5.1036057, [1].LeakTest.Detailed.element_data[7].Variable_code := 58, [1].LeakTest.Detailed.element_data[7].prec_code := 2, [1].LeakTest.Detailed.element_data[7].Unit_code := 60, [1].LeakTest.Detailed.element_data[7].result_measurement := -1.0002404, [1].LeakTest.Detailed.element_data[8].Variable_code := 59, [1].LeakTest.Detailed.element_data[8].prec_code := 2, [1].LeakTest.Detailed.element_data[8].Unit_code := 60, [1].LeakTest.Detailed.element_data[8].result_measurement := 1.0002404, [1].LeakTest.Detailed.element_data[9].Variable_code := 12, [1].LeakTest.Detailed.element_data[9].prec_code := 3, [1].LeakTest.Detailed.element_data[9].Unit_code := 12, [1].LeakTest.Detailed.element_data[9].result_measurement := 5.000001, [1].LeakTest.Detailed.element_data[10].Variable_code := 62, [1].LeakTest.Detailed.element_data[10].prec_code := 2, [1].LeakTest.Detailed.element_data[10].Unit_code := 60, [1].LeakTest.Detailed.element_data[10].result_measurement := 1.1002644, [1].LeakTest.Detailed.element_data[11].Variable_code := 21, [1].LeakTest.Detailed.element_data[11].prec_code := 3, [1].LeakTest.Detailed.element_data[11].Unit_code := 41, [1].LeakTest.Detailed.element_data[11].result_measurement := 0.0015180558, [1].LeakTest.Detailed.element_data[12].Variable_code := 25, [1].LeakTest.Detailed.element_data[12].prec_code := 3, [1].LeakTest.Detailed.element_data[12].Unit_code := 41, [1].LeakTest.Detailed.element_data[12].result_measurement := 0.021727756, [1].LeakTest.Detailed.element_data[13].Variable_code := 216, [1].LeakTest.Detailed.element_data[13].prec_code := 3, [1].LeakTest.Detailed.element_data[13].Unit_code := 41, [1].LeakTest.Detailed.element_data[13].result_measurement := 0.00085681677, [1].LeakTest.Detailed.element_data[14].Variable_code := 218, [1].LeakTest.Detailed.element_data[14].prec_code := 3, [1].LeakTest.Detailed.element_data[14].Unit_code := 41, [1].LeakTest.Detailed.element_data[14].result_measurement := 0.01094304, [1].LeakTest.Detailed.element_data[15].Variable_code := 295, [1].LeakTest.Detailed.element_data[15].prec_code := 3, [1].LeakTest.Detailed.element_data[15].Unit_code := 12, [1].LeakTest.Detailed.element_data[15].result_measurement := 5.1049933);
   DryCycle_N1Ready : BOOL;
   DryCycle_N2Ready : BOOL;
   DUTHistoryDump : udt_DUTHistory := (Barcode := 'A252620388', VolumeTest.UID := 25862, VolumeTest.Basic.unique_id := 25862, VolumeTest.Basic.channel_num := 1, VolumeTest.Basic.program_num := 1, VolumeTest.Basic.evaluation_code := 2, VolumeTest.Basic.test_port := 1, VolumeTest.Basic.year := 26, VolumeTest.Basic.month := 6, VolumeTest.Basic.date := 2, VolumeTest.Basic.hour := 14, VolumeTest.Basic.minute := 37, VolumeTest.Basic.second := 42, VolumeTest.Basic.flags := 12, VolumeTest.Basic.Num_tests := 1, VolumeTest.Basic.test_elements.test_type := 69, VolumeTest.Basic.test_elements.test_eval := 2, VolumeTest.Basic.test_elements.num_elements := 4, VolumeTest.Detailed.unique_id := 25862, VolumeTest.Detailed.num_elements := 4, VolumeTest.Detailed.Test_Type := 69, VolumeTest.Detailed.element_data[0].Variable_code := 245, VolumeTest.Detailed.element_data[0].prec_code := 2, VolumeTest.Detailed.element_data[0].Unit_code := 165, VolumeTest.Detailed.element_data[0].result_measurement := 214.21709, VolumeTest.Detailed.element_data[1].Variable_code := 13, VolumeTest.Detailed.element_data[1].prec_code := 3, VolumeTest.Detailed.element_data[1].Unit_code := 12, VolumeTest.Detailed.element_data[1].result_measurement := 1.5958865, VolumeTest.Detailed.element_data[2].Variable_code := 247, VolumeTest.Detailed.element_data[2].prec_code := 3, VolumeTest.Detailed.element_data[2].Unit_code := 12, VolumeTest.Detailed.element_data[2].result_measurement := 5.0145483, VolumeTest.Detailed.element_data[3].Variable_code := 295, VolumeTest.Detailed.element_data[3].prec_code := 3, VolumeTest.Detailed.element_data[3].Unit_code := 12, VolumeTest.Detailed.element_data[3].result_measurement := 5.0152373, LeakTest.Detailed.element_data[0].result_measurement := -999.0);
   DUTTestHistory : udt_DUTHistory[100] := ([0].Barcode := 'A252620388', [0].VolumeTest.UID := 25862, [0].VolumeTest.Basic.unique_id := 25862, [0].VolumeTest.Basic.channel_num := 1, [0].VolumeTest.Basic.program_num := 1, [0].VolumeTest.Basic.evaluation_code := 2, [0].VolumeTest.Basic.test_port := 1, [0].VolumeTest.Basic.year := 26, [0].VolumeTest.Basic.month := 6, [0].VolumeTest.Basic.date := 2, [0].VolumeTest.Basic.hour := 14, [0].VolumeTest.Basic.minute := 37, [0].VolumeTest.Basic.second := 42, [0].VolumeTest.Basic.flags := 12, [0].VolumeTest.Basic.Num_tests := 1, [0].VolumeTest.Basic.test_elements.test_type := 69, [0].VolumeTest.Basic.test_elements.test_eval := 2, [0].VolumeTest.Basic.test_elements.num_elements := 4, [0].VolumeTest.Detailed.unique_id := 25862, [0].VolumeTest.Detailed.num_elements := 4, [0].VolumeTest.Detailed.Test_Type := 69, [0].VolumeTest.Detailed.element_data[0].Variable_code := 245, [0].VolumeTest.Detailed.element_data[0].prec_code := 2, [0].VolumeTest.Detailed.element_data[0].Unit_code := 165, [0].VolumeTest.Detailed.element_data[0].result_measurement := 214.21709, [0].VolumeTest.Detailed.element_data[1].Variable_code := 13, [0].VolumeTest.Detailed.element_data[1].prec_code := 3, [0].VolumeTest.Detailed.element_data[1].Unit_code := 12, [0].VolumeTest.Detailed.element_data[1].result_measurement := 1.5958865, [0].VolumeTest.Detailed.element_data[2].Variable_code := 247, [0].VolumeTest.Detailed.element_data[2].prec_code := 3, [0].VolumeTest.Detailed.element_data[2].Unit_code := 12, [0].VolumeTest.Detailed.element_data[2].result_measurement := 5.0145483, [0].VolumeTest.Detailed.element_data[3].Variable_code := 295, [0].VolumeTest.Detailed.element_data[3].prec_code := 3, [0].VolumeTest.Detailed.element_data[3].Unit_code := 12, [0].VolumeTest.Detailed.element_data[3].result_measurement := 5.0152373, [0].LeakTest.Detailed.element_data[0].result_measurement := -999.0, [1].Barcode := 'A252620388', [1].VolumeTest.UID := 25862, [1].VolumeTest.Basic.unique_id := 25862, [1].VolumeTest.Basic.channel_num := 1, [1].VolumeTest.Basic.program_num := 1, [1].VolumeTest.Basic.evaluation_code := 2, [1].VolumeTest.Basic.test_port := 1, [1].VolumeTest.Basic.year := 26, [1].VolumeTest.Basic.month := 6, [1].VolumeTest.Basic.date := 2, [1].VolumeTest.Basic.hour := 14, [1].VolumeTest.Basic.minute := 37, [1].VolumeTest.Basic.second := 42, [1].VolumeTest.Basic.flags := 12, [1].VolumeTest.Basic.Num_tests := 1, [1].VolumeTest.Basic.test_elements.test_type := 69, [1].VolumeTest.Basic.test_elements.test_eval := 2, [1].VolumeTest.Basic.test_elements.num_elements := 4, [1].VolumeTest.Detailed.unique_id := 25862, [1].VolumeTest.Detailed.num_elements := 4, [1].VolumeTest.Detailed.Test_Type := 69, [1].VolumeTest.Detailed.element_data[0].Variable_code := 245,
        [1].VolumeTest.Detailed.element_data[0].prec_code := 2, [1].VolumeTest.Detailed.element_data[0].Unit_code := 165, [1].VolumeTest.Detailed.element_data[0].result_measurement := 214.21709, [1].VolumeTest.Detailed.element_data[1].Variable_code := 13, [1].VolumeTest.Detailed.element_data[1].prec_code := 3, [1].VolumeTest.Detailed.element_data[1].Unit_code := 12, [1].VolumeTest.Detailed.element_data[1].result_measurement := 1.5958865, [1].VolumeTest.Detailed.element_data[2].Variable_code := 247, [1].VolumeTest.Detailed.element_data[2].prec_code := 3, [1].VolumeTest.Detailed.element_data[2].Unit_code := 12, [1].VolumeTest.Detailed.element_data[2].result_measurement := 5.0145483, [1].VolumeTest.Detailed.element_data[3].Variable_code := 295, [1].VolumeTest.Detailed.element_data[3].prec_code := 3, [1].VolumeTest.Detailed.element_data[3].Unit_code := 12, [1].VolumeTest.Detailed.element_data[3].result_measurement := 5.0152373, [1].LeakTest.Detailed.element_data[0].result_measurement := -999.0, [2].Barcode := 'A252620388', [2].VolumeTest.UID := 25862, [2].VolumeTest.Basic.unique_id := 25862, [2].VolumeTest.Basic.channel_num := 1, [2].VolumeTest.Basic.program_num := 1, [2].VolumeTest.Basic.evaluation_code := 2, [2].VolumeTest.Basic.test_port := 1, [2].VolumeTest.Basic.year := 26, [2].VolumeTest.Basic.month := 6, [2].VolumeTest.Basic.date := 2, [2].VolumeTest.Basic.hour := 14, [2].VolumeTest.Basic.minute := 37, [2].VolumeTest.Basic.second := 42, [2].VolumeTest.Basic.flags := 12, [2].VolumeTest.Basic.Num_tests := 1, [2].VolumeTest.Basic.test_elements.test_type := 69, [2].VolumeTest.Basic.test_elements.test_eval := 2, [2].VolumeTest.Basic.test_elements.num_elements := 4, [2].VolumeTest.Detailed.unique_id := 25862, [2].VolumeTest.Detailed.num_elements := 4, [2].VolumeTest.Detailed.Test_Type := 69, [2].VolumeTest.Detailed.element_data[0].Variable_code := 245, [2].VolumeTest.Detailed.element_data[0].prec_code := 2, [2].VolumeTest.Detailed.element_data[0].Unit_code := 165, [2].VolumeTest.Detailed.element_data[0].result_measurement := 214.21709, [2].VolumeTest.Detailed.element_data[1].Variable_code := 13, [2].VolumeTest.Detailed.element_data[1].prec_code := 3, [2].VolumeTest.Detailed.element_data[1].Unit_code := 12, [2].VolumeTest.Detailed.element_data[1].result_measurement := 1.5958865, [2].VolumeTest.Detailed.element_data[2].Variable_code := 247, [2].VolumeTest.Detailed.element_data[2].prec_code := 3, [2].VolumeTest.Detailed.element_data[2].Unit_code := 12, [2].VolumeTest.Detailed.element_data[2].result_measurement := 5.0145483, [2].VolumeTest.Detailed.element_data[3].Variable_code := 295, [2].VolumeTest.Detailed.element_data[3].prec_code := 3, [2].VolumeTest.Detailed.element_data[3].Unit_code := 12, [2].VolumeTest.Detailed.element_data[3].result_measurement := 5.0152373, [2].LeakTest.Detailed.element_data[0].result_measurement := -999.0, [3].Barcode := 'A252620388', [3].VolumeTest.UID := 25862, [3].VolumeTest.Basic.unique_id := 25862, [3].VolumeTest.Basic.channel_num := 1, [3].VolumeTest.Basic.program_num := 1, [3].VolumeTest.Basic.evaluation_code := 2,
        [3].VolumeTest.Basic.test_port := 1, [3].VolumeTest.Basic.year := 26, [3].VolumeTest.Basic.month := 6, [3].VolumeTest.Basic.date := 2, [3].VolumeTest.Basic.hour := 14, [3].VolumeTest.Basic.minute := 37, [3].VolumeTest.Basic.second := 42, [3].VolumeTest.Basic.flags := 12, [3].VolumeTest.Basic.Num_tests := 1, [3].VolumeTest.Basic.test_elements.test_type := 69, [3].VolumeTest.Basic.test_elements.test_eval := 2, [3].VolumeTest.Basic.test_elements.num_elements := 4, [3].VolumeTest.Detailed.unique_id := 25862, [3].VolumeTest.Detailed.num_elements := 4, [3].VolumeTest.Detailed.Test_Type := 69, [3].VolumeTest.Detailed.element_data[0].Variable_code := 245, [3].VolumeTest.Detailed.element_data[0].prec_code := 2, [3].VolumeTest.Detailed.element_data[0].Unit_code := 165, [3].VolumeTest.Detailed.element_data[0].result_measurement := 214.21709, [3].VolumeTest.Detailed.element_data[1].Variable_code := 13, [3].VolumeTest.Detailed.element_data[1].prec_code := 3, [3].VolumeTest.Detailed.element_data[1].Unit_code := 12, [3].VolumeTest.Detailed.element_data[1].result_measurement := 1.5958865, [3].VolumeTest.Detailed.element_data[2].Variable_code := 247, [3].VolumeTest.Detailed.element_data[2].prec_code := 3, [3].VolumeTest.Detailed.element_data[2].Unit_code := 12, [3].VolumeTest.Detailed.element_data[2].result_measurement := 5.0145483, [3].VolumeTest.Detailed.element_data[3].Variable_code := 295, [3].VolumeTest.Detailed.element_data[3].prec_code := 3, [3].VolumeTest.Detailed.element_data[3].Unit_code := 12, [3].VolumeTest.Detailed.element_data[3].result_measurement := 5.0152373, [3].LeakTest.Detailed.element_data[0].result_measurement := -999.0, [4].Barcode := 'A252620388', [4].VolumeTest.UID := 25862, [4].VolumeTest.Basic.unique_id := 25862, [4].VolumeTest.Basic.channel_num := 1, [4].VolumeTest.Basic.program_num := 1, [4].VolumeTest.Basic.evaluation_code := 2, [4].VolumeTest.Basic.test_port := 1, [4].VolumeTest.Basic.year := 26, [4].VolumeTest.Basic.month := 6, [4].VolumeTest.Basic.date := 2, [4].VolumeTest.Basic.hour := 14, [4].VolumeTest.Basic.minute := 37, [4].VolumeTest.Basic.second := 42, [4].VolumeTest.Basic.flags := 12, [4].VolumeTest.Basic.Num_tests := 1, [4].VolumeTest.Basic.test_elements.test_type := 69, [4].VolumeTest.Basic.test_elements.test_eval := 2, [4].VolumeTest.Basic.test_elements.num_elements := 4, [4].VolumeTest.Detailed.unique_id := 25862, [4].VolumeTest.Detailed.num_elements := 4, [4].VolumeTest.Detailed.Test_Type := 69, [4].VolumeTest.Detailed.element_data[0].Variable_code := 245, [4].VolumeTest.Detailed.element_data[0].prec_code := 2, [4].VolumeTest.Detailed.element_data[0].Unit_code := 165, [4].VolumeTest.Detailed.element_data[0].result_measurement := 214.21709, [4].VolumeTest.Detailed.element_data[1].Variable_code := 13, [4].VolumeTest.Detailed.element_data[1].prec_code := 3, [4].VolumeTest.Detailed.element_data[1].Unit_code := 12,
        [4].VolumeTest.Detailed.element_data[1].result_measurement := 1.5958865, [4].VolumeTest.Detailed.element_data[2].Variable_code := 247, [4].VolumeTest.Detailed.element_data[2].prec_code := 3, [4].VolumeTest.Detailed.element_data[2].Unit_code := 12, [4].VolumeTest.Detailed.element_data[2].result_measurement := 5.0145483, [4].VolumeTest.Detailed.element_data[3].Variable_code := 295, [4].VolumeTest.Detailed.element_data[3].prec_code := 3, [4].VolumeTest.Detailed.element_data[3].Unit_code := 12, [4].VolumeTest.Detailed.element_data[3].result_measurement := 5.0152373, [4].LeakTest.Detailed.element_data[0].result_measurement := -999.0, [5].Barcode := 'A252620388', [5].VolumeTest.UID := 25862, [5].VolumeTest.Basic.unique_id := 25862, [5].VolumeTest.Basic.channel_num := 1, [5].VolumeTest.Basic.program_num := 1, [5].VolumeTest.Basic.evaluation_code := 2, [5].VolumeTest.Basic.test_port := 1, [5].VolumeTest.Basic.year := 26, [5].VolumeTest.Basic.month := 6, [5].VolumeTest.Basic.date := 2, [5].VolumeTest.Basic.hour := 14, [5].VolumeTest.Basic.minute := 37, [5].VolumeTest.Basic.second := 42, [5].VolumeTest.Basic.flags := 12, [5].VolumeTest.Basic.Num_tests := 1, [5].VolumeTest.Basic.test_elements.test_type := 69, [5].VolumeTest.Basic.test_elements.test_eval := 2, [5].VolumeTest.Basic.test_elements.num_elements := 4, [5].VolumeTest.Detailed.unique_id := 25862, [5].VolumeTest.Detailed.num_elements := 4, [5].VolumeTest.Detailed.Test_Type := 69, [5].VolumeTest.Detailed.element_data[0].Variable_code := 245, [5].VolumeTest.Detailed.element_data[0].prec_code := 2, [5].VolumeTest.Detailed.element_data[0].Unit_code := 165, [5].VolumeTest.Detailed.element_data[0].result_measurement := 214.21709, [5].VolumeTest.Detailed.element_data[1].Variable_code := 13, [5].VolumeTest.Detailed.element_data[1].prec_code := 3, [5].VolumeTest.Detailed.element_data[1].Unit_code := 12, [5].VolumeTest.Detailed.element_data[1].result_measurement := 1.5958865, [5].VolumeTest.Detailed.element_data[2].Variable_code := 247, [5].VolumeTest.Detailed.element_data[2].prec_code := 3, [5].VolumeTest.Detailed.element_data[2].Unit_code := 12, [5].VolumeTest.Detailed.element_data[2].result_measurement := 5.0145483, [5].VolumeTest.Detailed.element_data[3].Variable_code := 295, [5].VolumeTest.Detailed.element_data[3].prec_code := 3, [5].VolumeTest.Detailed.element_data[3].Unit_code := 12, [5].VolumeTest.Detailed.element_data[3].result_measurement := 5.0152373, [5].LeakTest.Detailed.element_data[0].result_measurement := -999.0, [6].Barcode := 'A252620388', [6].VolumeTest.UID := 25862, [6].VolumeTest.Basic.unique_id := 25862, [6].VolumeTest.Basic.channel_num := 1, [6].VolumeTest.Basic.program_num := 1, [6].VolumeTest.Basic.evaluation_code := 2, [6].VolumeTest.Basic.test_port := 1, [6].VolumeTest.Basic.year := 26, [6].VolumeTest.Basic.month := 6, [6].VolumeTest.Basic.date := 2, [6].VolumeTest.Basic.hour := 14, [6].VolumeTest.Basic.minute := 37,
        [6].VolumeTest.Basic.second := 42, [6].VolumeTest.Basic.flags := 12, [6].VolumeTest.Basic.Num_tests := 1, [6].VolumeTest.Basic.test_elements.test_type := 69, [6].VolumeTest.Basic.test_elements.test_eval := 2, [6].VolumeTest.Basic.test_elements.num_elements := 4, [6].VolumeTest.Detailed.unique_id := 25862, [6].VolumeTest.Detailed.num_elements := 4, [6].VolumeTest.Detailed.Test_Type := 69, [6].VolumeTest.Detailed.element_data[0].Variable_code := 245, [6].VolumeTest.Detailed.element_data[0].prec_code := 2, [6].VolumeTest.Detailed.element_data[0].Unit_code := 165, [6].VolumeTest.Detailed.element_data[0].result_measurement := 214.21709, [6].VolumeTest.Detailed.element_data[1].Variable_code := 13, [6].VolumeTest.Detailed.element_data[1].prec_code := 3, [6].VolumeTest.Detailed.element_data[1].Unit_code := 12, [6].VolumeTest.Detailed.element_data[1].result_measurement := 1.5958865, [6].VolumeTest.Detailed.element_data[2].Variable_code := 247, [6].VolumeTest.Detailed.element_data[2].prec_code := 3, [6].VolumeTest.Detailed.element_data[2].Unit_code := 12, [6].VolumeTest.Detailed.element_data[2].result_measurement := 5.0145483, [6].VolumeTest.Detailed.element_data[3].Variable_code := 295, [6].VolumeTest.Detailed.element_data[3].prec_code := 3, [6].VolumeTest.Detailed.element_data[3].Unit_code := 12, [6].VolumeTest.Detailed.element_data[3].result_measurement := 5.0152373, [6].LeakTest.Detailed.element_data[0].result_measurement := -999.0, [7].Barcode := 'A252620388', [7].VolumeTest.UID := 25862, [7].VolumeTest.Basic.unique_id := 25862, [7].VolumeTest.Basic.channel_num := 1, [7].VolumeTest.Basic.program_num := 1, [7].VolumeTest.Basic.evaluation_code := 2, [7].VolumeTest.Basic.test_port := 1, [7].VolumeTest.Basic.year := 26, [7].VolumeTest.Basic.month := 6, [7].VolumeTest.Basic.date := 2, [7].VolumeTest.Basic.hour := 14, [7].VolumeTest.Basic.minute := 37, [7].VolumeTest.Basic.second := 42, [7].VolumeTest.Basic.flags := 12, [7].VolumeTest.Basic.Num_tests := 1, [7].VolumeTest.Basic.test_elements.test_type := 69, [7].VolumeTest.Basic.test_elements.test_eval := 2, [7].VolumeTest.Basic.test_elements.num_elements := 4, [7].VolumeTest.Detailed.unique_id := 25862, [7].VolumeTest.Detailed.num_elements := 4, [7].VolumeTest.Detailed.Test_Type := 69, [7].VolumeTest.Detailed.element_data[0].Variable_code := 245, [7].VolumeTest.Detailed.element_data[0].prec_code := 2, [7].VolumeTest.Detailed.element_data[0].Unit_code := 165, [7].VolumeTest.Detailed.element_data[0].result_measurement := 214.21709, [7].VolumeTest.Detailed.element_data[1].Variable_code := 13, [7].VolumeTest.Detailed.element_data[1].prec_code := 3, [7].VolumeTest.Detailed.element_data[1].Unit_code := 12, [7].VolumeTest.Detailed.element_data[1].result_measurement := 1.5958865, [7].VolumeTest.Detailed.element_data[2].Variable_code := 247, [7].VolumeTest.Detailed.element_data[2].prec_code := 3, [7].VolumeTest.Detailed.element_data[2].Unit_code := 12, [7].VolumeTest.Detailed.element_data[2].result_measurement := 5.0145483, [7].VolumeTest.Detailed.element_data[3].Variable_code := 295,
        [7].VolumeTest.Detailed.element_data[3].prec_code := 3, [7].VolumeTest.Detailed.element_data[3].Unit_code := 12, [7].VolumeTest.Detailed.element_data[3].result_measurement := 5.0152373, [7].LeakTest.Detailed.element_data[0].result_measurement := -999.0, [8].Barcode := 'A252620388', [8].VolumeTest.UID := 25862, [8].VolumeTest.Basic.unique_id := 25862, [8].VolumeTest.Basic.channel_num := 1, [8].VolumeTest.Basic.program_num := 1, [8].VolumeTest.Basic.evaluation_code := 2, [8].VolumeTest.Basic.test_port := 1, [8].VolumeTest.Basic.year := 26, [8].VolumeTest.Basic.month := 6, [8].VolumeTest.Basic.date := 2, [8].VolumeTest.Basic.hour := 14, [8].VolumeTest.Basic.minute := 37, [8].VolumeTest.Basic.second := 42, [8].VolumeTest.Basic.flags := 12, [8].VolumeTest.Basic.Num_tests := 1, [8].VolumeTest.Basic.test_elements.test_type := 69, [8].VolumeTest.Basic.test_elements.test_eval := 2, [8].VolumeTest.Basic.test_elements.num_elements := 4, [8].VolumeTest.Detailed.unique_id := 25862, [8].VolumeTest.Detailed.num_elements := 4, [8].VolumeTest.Detailed.Test_Type := 69, [8].VolumeTest.Detailed.element_data[0].Variable_code := 245, [8].VolumeTest.Detailed.element_data[0].prec_code := 2, [8].VolumeTest.Detailed.element_data[0].Unit_code := 165, [8].VolumeTest.Detailed.element_data[0].result_measurement := 214.21709, [8].VolumeTest.Detailed.element_data[1].Variable_code := 13, [8].VolumeTest.Detailed.element_data[1].prec_code := 3, [8].VolumeTest.Detailed.element_data[1].Unit_code := 12, [8].VolumeTest.Detailed.element_data[1].result_measurement := 1.5958865, [8].VolumeTest.Detailed.element_data[2].Variable_code := 247, [8].VolumeTest.Detailed.element_data[2].prec_code := 3, [8].VolumeTest.Detailed.element_data[2].Unit_code := 12, [8].VolumeTest.Detailed.element_data[2].result_measurement := 5.0145483, [8].VolumeTest.Detailed.element_data[3].Variable_code := 295, [8].VolumeTest.Detailed.element_data[3].prec_code := 3, [8].VolumeTest.Detailed.element_data[3].Unit_code := 12, [8].VolumeTest.Detailed.element_data[3].result_measurement := 5.0152373, [8].LeakTest.Detailed.element_data[0].result_measurement := -999.0, [9].Barcode := 'A252620388', [9].VolumeTest.UID := 25862, [9].VolumeTest.Basic.unique_id := 25862, [9].VolumeTest.Basic.channel_num := 1, [9].VolumeTest.Basic.program_num := 1, [9].VolumeTest.Basic.evaluation_code := 2, [9].VolumeTest.Basic.test_port := 1, [9].VolumeTest.Basic.year := 26, [9].VolumeTest.Basic.month := 6, [9].VolumeTest.Basic.date := 2, [9].VolumeTest.Basic.hour := 14, [9].VolumeTest.Basic.minute := 37, [9].VolumeTest.Basic.second := 42, [9].VolumeTest.Basic.flags := 12, [9].VolumeTest.Basic.Num_tests := 1, [9].VolumeTest.Basic.test_elements.test_type := 69, [9].VolumeTest.Basic.test_elements.test_eval := 2, [9].VolumeTest.Basic.test_elements.num_elements := 4,
        [9].VolumeTest.Detailed.unique_id := 25862, [9].VolumeTest.Detailed.num_elements := 4, [9].VolumeTest.Detailed.Test_Type := 69, [9].VolumeTest.Detailed.element_data[0].Variable_code := 245, [9].VolumeTest.Detailed.element_data[0].prec_code := 2, [9].VolumeTest.Detailed.element_data[0].Unit_code := 165, [9].VolumeTest.Detailed.element_data[0].result_measurement := 214.21709, [9].VolumeTest.Detailed.element_data[1].Variable_code := 13, [9].VolumeTest.Detailed.element_data[1].prec_code := 3, [9].VolumeTest.Detailed.element_data[1].Unit_code := 12, [9].VolumeTest.Detailed.element_data[1].result_measurement := 1.5958865, [9].VolumeTest.Detailed.element_data[2].Variable_code := 247, [9].VolumeTest.Detailed.element_data[2].prec_code := 3, [9].VolumeTest.Detailed.element_data[2].Unit_code := 12, [9].VolumeTest.Detailed.element_data[2].result_measurement := 5.0145483, [9].VolumeTest.Detailed.element_data[3].Variable_code := 295, [9].VolumeTest.Detailed.element_data[3].prec_code := 3, [9].VolumeTest.Detailed.element_data[3].Unit_code := 12, [9].VolumeTest.Detailed.element_data[3].result_measurement := 5.0152373, [9].LeakTest.Detailed.element_data[0].result_measurement := -999.0, [10].Barcode := 'A252620388', [10].VolumeTest.UID := 25862, [10].VolumeTest.Basic.unique_id := 25862, [10].VolumeTest.Basic.channel_num := 1, [10].VolumeTest.Basic.program_num := 1, [10].VolumeTest.Basic.evaluation_code := 2, [10].VolumeTest.Basic.test_port := 1, [10].VolumeTest.Basic.year := 26, [10].VolumeTest.Basic.month := 6, [10].VolumeTest.Basic.date := 2, [10].VolumeTest.Basic.hour := 14, [10].VolumeTest.Basic.minute := 37, [10].VolumeTest.Basic.second := 42, [10].VolumeTest.Basic.flags := 12, [10].VolumeTest.Basic.Num_tests := 1, [10].VolumeTest.Basic.test_elements.test_type := 69, [10].VolumeTest.Basic.test_elements.test_eval := 2, [10].VolumeTest.Basic.test_elements.num_elements := 4, [10].VolumeTest.Detailed.unique_id := 25862, [10].VolumeTest.Detailed.num_elements := 4, [10].VolumeTest.Detailed.Test_Type := 69, [10].VolumeTest.Detailed.element_data[0].Variable_code := 245, [10].VolumeTest.Detailed.element_data[0].prec_code := 2, [10].VolumeTest.Detailed.element_data[0].Unit_code := 165, [10].VolumeTest.Detailed.element_data[0].result_measurement := 214.21709, [10].VolumeTest.Detailed.element_data[1].Variable_code := 13, [10].VolumeTest.Detailed.element_data[1].prec_code := 3, [10].VolumeTest.Detailed.element_data[1].Unit_code := 12, [10].VolumeTest.Detailed.element_data[1].result_measurement := 1.5958865, [10].VolumeTest.Detailed.element_data[2].Variable_code := 247, [10].VolumeTest.Detailed.element_data[2].prec_code := 3, [10].VolumeTest.Detailed.element_data[2].Unit_code := 12, [10].VolumeTest.Detailed.element_data[2].result_measurement := 5.0145483, [10].VolumeTest.Detailed.element_data[3].Variable_code := 295, [10].VolumeTest.Detailed.element_data[3].prec_code := 3, [10].VolumeTest.Detailed.element_data[3].Unit_code := 12, [10].VolumeTest.Detailed.element_data[3].result_measurement := 5.0152373, [10].LeakTest.Detailed.element_data[0].result_measurement := -999.0, [11].Barcode := 'A252620388', [11].VolumeTest.UID := 25862,
        [11].VolumeTest.Basic.unique_id := 25862, [11].VolumeTest.Basic.channel_num := 1, [11].VolumeTest.Basic.program_num := 1, [11].VolumeTest.Basic.evaluation_code := 2, [11].VolumeTest.Basic.test_port := 1, [11].VolumeTest.Basic.year := 26, [11].VolumeTest.Basic.month := 6, [11].VolumeTest.Basic.date := 2, [11].VolumeTest.Basic.hour := 14, [11].VolumeTest.Basic.minute := 37, [11].VolumeTest.Basic.second := 42, [11].VolumeTest.Basic.flags := 12, [11].VolumeTest.Basic.Num_tests := 1, [11].VolumeTest.Basic.test_elements.test_type := 69, [11].VolumeTest.Basic.test_elements.test_eval := 2, [11].VolumeTest.Basic.test_elements.num_elements := 4, [11].VolumeTest.Detailed.unique_id := 25862, [11].VolumeTest.Detailed.num_elements := 4, [11].VolumeTest.Detailed.Test_Type := 69, [11].VolumeTest.Detailed.element_data[0].Variable_code := 245, [11].VolumeTest.Detailed.element_data[0].prec_code := 2, [11].VolumeTest.Detailed.element_data[0].Unit_code := 165, [11].VolumeTest.Detailed.element_data[0].result_measurement := 214.21709, [11].VolumeTest.Detailed.element_data[1].Variable_code := 13, [11].VolumeTest.Detailed.element_data[1].prec_code := 3, [11].VolumeTest.Detailed.element_data[1].Unit_code := 12, [11].VolumeTest.Detailed.element_data[1].result_measurement := 1.5958865, [11].VolumeTest.Detailed.element_data[2].Variable_code := 247, [11].VolumeTest.Detailed.element_data[2].prec_code := 3, [11].VolumeTest.Detailed.element_data[2].Unit_code := 12, [11].VolumeTest.Detailed.element_data[2].result_measurement := 5.0145483, [11].VolumeTest.Detailed.element_data[3].Variable_code := 295, [11].VolumeTest.Detailed.element_data[3].prec_code := 3, [11].VolumeTest.Detailed.element_data[3].Unit_code := 12, [11].VolumeTest.Detailed.element_data[3].result_measurement := 5.0152373, [11].LeakTest.Detailed.element_data[0].result_measurement := -999.0, [12].Barcode := 'A252620388', [12].VolumeTest.UID := 25862, [12].VolumeTest.Basic.unique_id := 25862, [12].VolumeTest.Basic.channel_num := 1, [12].VolumeTest.Basic.program_num := 1, [12].VolumeTest.Basic.evaluation_code := 2, [12].VolumeTest.Basic.test_port := 1, [12].VolumeTest.Basic.year := 26, [12].VolumeTest.Basic.month := 6, [12].VolumeTest.Basic.date := 2, [12].VolumeTest.Basic.hour := 14, [12].VolumeTest.Basic.minute := 37, [12].VolumeTest.Basic.second := 42, [12].VolumeTest.Basic.flags := 12, [12].VolumeTest.Basic.Num_tests := 1, [12].VolumeTest.Basic.test_elements.test_type := 69, [12].VolumeTest.Basic.test_elements.test_eval := 2, [12].VolumeTest.Basic.test_elements.num_elements := 4, [12].VolumeTest.Detailed.unique_id := 25862, [12].VolumeTest.Detailed.num_elements := 4, [12].VolumeTest.Detailed.Test_Type := 69, [12].VolumeTest.Detailed.element_data[0].Variable_code := 245, [12].VolumeTest.Detailed.element_data[0].prec_code := 2, [12].VolumeTest.Detailed.element_data[0].Unit_code := 165,
        [12].VolumeTest.Detailed.element_data[0].result_measurement := 214.21709, [12].VolumeTest.Detailed.element_data[1].Variable_code := 13, [12].VolumeTest.Detailed.element_data[1].prec_code := 3, [12].VolumeTest.Detailed.element_data[1].Unit_code := 12, [12].VolumeTest.Detailed.element_data[1].result_measurement := 1.5958865, [12].VolumeTest.Detailed.element_data[2].Variable_code := 247, [12].VolumeTest.Detailed.element_data[2].prec_code := 3, [12].VolumeTest.Detailed.element_data[2].Unit_code := 12, [12].VolumeTest.Detailed.element_data[2].result_measurement := 5.0145483, [12].VolumeTest.Detailed.element_data[3].Variable_code := 295, [12].VolumeTest.Detailed.element_data[3].prec_code := 3, [12].VolumeTest.Detailed.element_data[3].Unit_code := 12, [12].VolumeTest.Detailed.element_data[3].result_measurement := 5.0152373, [12].LeakTest.Detailed.element_data[0].result_measurement := -999.0, [13].Barcode := 'A252620388', [13].VolumeTest.UID := 25862, [13].VolumeTest.Basic.unique_id := 25862, [13].VolumeTest.Basic.channel_num := 1, [13].VolumeTest.Basic.program_num := 1, [13].VolumeTest.Basic.evaluation_code := 2, [13].VolumeTest.Basic.test_port := 1, [13].VolumeTest.Basic.year := 26, [13].VolumeTest.Basic.month := 6, [13].VolumeTest.Basic.date := 2, [13].VolumeTest.Basic.hour := 14, [13].VolumeTest.Basic.minute := 37, [13].VolumeTest.Basic.second := 42, [13].VolumeTest.Basic.flags := 12, [13].VolumeTest.Basic.Num_tests := 1, [13].VolumeTest.Basic.test_elements.test_type := 69, [13].VolumeTest.Basic.test_elements.test_eval := 2, [13].VolumeTest.Basic.test_elements.num_elements := 4, [13].VolumeTest.Detailed.unique_id := 25862, [13].VolumeTest.Detailed.num_elements := 4, [13].VolumeTest.Detailed.Test_Type := 69, [13].VolumeTest.Detailed.element_data[0].Variable_code := 245, [13].VolumeTest.Detailed.element_data[0].prec_code := 2, [13].VolumeTest.Detailed.element_data[0].Unit_code := 165, [13].VolumeTest.Detailed.element_data[0].result_measurement := 214.21709, [13].VolumeTest.Detailed.element_data[1].Variable_code := 13, [13].VolumeTest.Detailed.element_data[1].prec_code := 3, [13].VolumeTest.Detailed.element_data[1].Unit_code := 12, [13].VolumeTest.Detailed.element_data[1].result_measurement := 1.5958865, [13].VolumeTest.Detailed.element_data[2].Variable_code := 247, [13].VolumeTest.Detailed.element_data[2].prec_code := 3, [13].VolumeTest.Detailed.element_data[2].Unit_code := 12, [13].VolumeTest.Detailed.element_data[2].result_measurement := 5.0145483, [13].VolumeTest.Detailed.element_data[3].Variable_code := 295, [13].VolumeTest.Detailed.element_data[3].prec_code := 3, [13].VolumeTest.Detailed.element_data[3].Unit_code := 12, [13].VolumeTest.Detailed.element_data[3].result_measurement := 5.0152373, [13].LeakTest.Detailed.element_data[0].result_measurement := -999.0, [14].Barcode := 'A252620388', [14].VolumeTest.UID := 25862, [14].VolumeTest.Basic.unique_id := 25862, [14].VolumeTest.Basic.channel_num := 1, [14].VolumeTest.Basic.program_num := 1, [14].VolumeTest.Basic.evaluation_code := 2, [14].VolumeTest.Basic.test_port := 1, [14].VolumeTest.Basic.year := 26,
        [14].VolumeTest.Basic.month := 6, [14].VolumeTest.Basic.date := 2, [14].VolumeTest.Basic.hour := 14, [14].VolumeTest.Basic.minute := 37, [14].VolumeTest.Basic.second := 42, [14].VolumeTest.Basic.flags := 12, [14].VolumeTest.Basic.Num_tests := 1, [14].VolumeTest.Basic.test_elements.test_type := 69, [14].VolumeTest.Basic.test_elements.test_eval := 2, [14].VolumeTest.Basic.test_elements.num_elements := 4, [14].VolumeTest.Detailed.unique_id := 25862, [14].VolumeTest.Detailed.num_elements := 4, [14].VolumeTest.Detailed.Test_Type := 69, [14].VolumeTest.Detailed.element_data[0].Variable_code := 245, [14].VolumeTest.Detailed.element_data[0].prec_code := 2, [14].VolumeTest.Detailed.element_data[0].Unit_code := 165, [14].VolumeTest.Detailed.element_data[0].result_measurement := 214.21709, [14].VolumeTest.Detailed.element_data[1].Variable_code := 13, [14].VolumeTest.Detailed.element_data[1].prec_code := 3, [14].VolumeTest.Detailed.element_data[1].Unit_code := 12, [14].VolumeTest.Detailed.element_data[1].result_measurement := 1.5958865, [14].VolumeTest.Detailed.element_data[2].Variable_code := 247, [14].VolumeTest.Detailed.element_data[2].prec_code := 3, [14].VolumeTest.Detailed.element_data[2].Unit_code := 12, [14].VolumeTest.Detailed.element_data[2].result_measurement := 5.0145483, [14].VolumeTest.Detailed.element_data[3].Variable_code := 295, [14].VolumeTest.Detailed.element_data[3].prec_code := 3, [14].VolumeTest.Detailed.element_data[3].Unit_code := 12, [14].VolumeTest.Detailed.element_data[3].result_measurement := 5.0152373, [14].LeakTest.Detailed.element_data[0].result_measurement := -999.0, [15].Barcode := 'A252620388', [15].VolumeTest.UID := 25862, [15].VolumeTest.Basic.unique_id := 25862, [15].VolumeTest.Basic.channel_num := 1, [15].VolumeTest.Basic.program_num := 1, [15].VolumeTest.Basic.evaluation_code := 2, [15].VolumeTest.Basic.test_port := 1, [15].VolumeTest.Basic.year := 26, [15].VolumeTest.Basic.month := 6, [15].VolumeTest.Basic.date := 2, [15].VolumeTest.Basic.hour := 14, [15].VolumeTest.Basic.minute := 37, [15].VolumeTest.Basic.second := 42, [15].VolumeTest.Basic.flags := 12, [15].VolumeTest.Basic.Num_tests := 1, [15].VolumeTest.Basic.test_elements.test_type := 69, [15].VolumeTest.Basic.test_elements.test_eval := 2, [15].VolumeTest.Basic.test_elements.num_elements := 4, [15].VolumeTest.Detailed.unique_id := 25862, [15].VolumeTest.Detailed.num_elements := 4, [15].VolumeTest.Detailed.Test_Type := 69, [15].VolumeTest.Detailed.element_data[0].Variable_code := 245, [15].VolumeTest.Detailed.element_data[0].prec_code := 2, [15].VolumeTest.Detailed.element_data[0].Unit_code := 165, [15].VolumeTest.Detailed.element_data[0].result_measurement := 214.21709, [15].VolumeTest.Detailed.element_data[1].Variable_code := 13, [15].VolumeTest.Detailed.element_data[1].prec_code := 3, [15].VolumeTest.Detailed.element_data[1].Unit_code := 12, [15].VolumeTest.Detailed.element_data[1].result_measurement := 1.5958865, [15].VolumeTest.Detailed.element_data[2].Variable_code := 247,
        [15].VolumeTest.Detailed.element_data[2].prec_code := 3, [15].VolumeTest.Detailed.element_data[2].Unit_code := 12, [15].VolumeTest.Detailed.element_data[2].result_measurement := 5.0145483, [15].VolumeTest.Detailed.element_data[3].Variable_code := 295, [15].VolumeTest.Detailed.element_data[3].prec_code := 3, [15].VolumeTest.Detailed.element_data[3].Unit_code := 12, [15].VolumeTest.Detailed.element_data[3].result_measurement := 5.0152373, [15].LeakTest.Detailed.element_data[0].result_measurement := -999.0, [16].Barcode := 'A252620388', [16].VolumeTest.UID := 25862, [16].VolumeTest.Basic.unique_id := 25862, [16].VolumeTest.Basic.channel_num := 1, [16].VolumeTest.Basic.program_num := 1, [16].VolumeTest.Basic.evaluation_code := 2, [16].VolumeTest.Basic.test_port := 1, [16].VolumeTest.Basic.year := 26, [16].VolumeTest.Basic.month := 6, [16].VolumeTest.Basic.date := 2, [16].VolumeTest.Basic.hour := 14, [16].VolumeTest.Basic.minute := 37, [16].VolumeTest.Basic.second := 42, [16].VolumeTest.Basic.flags := 12, [16].VolumeTest.Basic.Num_tests := 1, [16].VolumeTest.Basic.test_elements.test_type := 69, [16].VolumeTest.Basic.test_elements.test_eval := 2, [16].VolumeTest.Basic.test_elements.num_elements := 4, [16].VolumeTest.Detailed.unique_id := 25862, [16].VolumeTest.Detailed.num_elements := 4, [16].VolumeTest.Detailed.Test_Type := 69, [16].VolumeTest.Detailed.element_data[0].Variable_code := 245, [16].VolumeTest.Detailed.element_data[0].prec_code := 2, [16].VolumeTest.Detailed.element_data[0].Unit_code := 165, [16].VolumeTest.Detailed.element_data[0].result_measurement := 214.21709, [16].VolumeTest.Detailed.element_data[1].Variable_code := 13, [16].VolumeTest.Detailed.element_data[1].prec_code := 3, [16].VolumeTest.Detailed.element_data[1].Unit_code := 12, [16].VolumeTest.Detailed.element_data[1].result_measurement := 1.5958865, [16].VolumeTest.Detailed.element_data[2].Variable_code := 247, [16].VolumeTest.Detailed.element_data[2].prec_code := 3, [16].VolumeTest.Detailed.element_data[2].Unit_code := 12, [16].VolumeTest.Detailed.element_data[2].result_measurement := 5.0145483, [16].VolumeTest.Detailed.element_data[3].Variable_code := 295, [16].VolumeTest.Detailed.element_data[3].prec_code := 3, [16].VolumeTest.Detailed.element_data[3].Unit_code := 12, [16].VolumeTest.Detailed.element_data[3].result_measurement := 5.0152373, [16].LeakTest.Detailed.element_data[0].result_measurement := -999.0, [17].Barcode := 'A252620388', [17].VolumeTest.UID := 25862, [17].VolumeTest.Basic.unique_id := 25862, [17].VolumeTest.Basic.channel_num := 1, [17].VolumeTest.Basic.program_num := 1, [17].VolumeTest.Basic.evaluation_code := 2, [17].VolumeTest.Basic.test_port := 1, [17].VolumeTest.Basic.year := 26, [17].VolumeTest.Basic.month := 6, [17].VolumeTest.Basic.date := 2, [17].VolumeTest.Basic.hour := 14, [17].VolumeTest.Basic.minute := 37, [17].VolumeTest.Basic.second := 42, [17].VolumeTest.Basic.flags := 12,
        [17].VolumeTest.Basic.Num_tests := 1, [17].VolumeTest.Basic.test_elements.test_type := 69, [17].VolumeTest.Basic.test_elements.test_eval := 2, [17].VolumeTest.Basic.test_elements.num_elements := 4, [17].VolumeTest.Detailed.unique_id := 25862, [17].VolumeTest.Detailed.num_elements := 4, [17].VolumeTest.Detailed.Test_Type := 69, [17].VolumeTest.Detailed.element_data[0].Variable_code := 245, [17].VolumeTest.Detailed.element_data[0].prec_code := 2, [17].VolumeTest.Detailed.element_data[0].Unit_code := 165, [17].VolumeTest.Detailed.element_data[0].result_measurement := 214.21709, [17].VolumeTest.Detailed.element_data[1].Variable_code := 13, [17].VolumeTest.Detailed.element_data[1].prec_code := 3, [17].VolumeTest.Detailed.element_data[1].Unit_code := 12, [17].VolumeTest.Detailed.element_data[1].result_measurement := 1.5958865, [17].VolumeTest.Detailed.element_data[2].Variable_code := 247, [17].VolumeTest.Detailed.element_data[2].prec_code := 3, [17].VolumeTest.Detailed.element_data[2].Unit_code := 12, [17].VolumeTest.Detailed.element_data[2].result_measurement := 5.0145483, [17].VolumeTest.Detailed.element_data[3].Variable_code := 295, [17].VolumeTest.Detailed.element_data[3].prec_code := 3, [17].VolumeTest.Detailed.element_data[3].Unit_code := 12, [17].VolumeTest.Detailed.element_data[3].result_measurement := 5.0152373, [17].LeakTest.Detailed.element_data[0].result_measurement := -999.0, [18].Barcode := 'A252620388', [18].VolumeTest.UID := 25862, [18].VolumeTest.Basic.unique_id := 25862, [18].VolumeTest.Basic.channel_num := 1, [18].VolumeTest.Basic.program_num := 1, [18].VolumeTest.Basic.evaluation_code := 2, [18].VolumeTest.Basic.test_port := 1, [18].VolumeTest.Basic.year := 26, [18].VolumeTest.Basic.month := 6, [18].VolumeTest.Basic.date := 2, [18].VolumeTest.Basic.hour := 14, [18].VolumeTest.Basic.minute := 37, [18].VolumeTest.Basic.second := 42, [18].VolumeTest.Basic.flags := 12, [18].VolumeTest.Basic.Num_tests := 1, [18].VolumeTest.Basic.test_elements.test_type := 69, [18].VolumeTest.Basic.test_elements.test_eval := 2, [18].VolumeTest.Basic.test_elements.num_elements := 4, [18].VolumeTest.Detailed.unique_id := 25862, [18].VolumeTest.Detailed.num_elements := 4, [18].VolumeTest.Detailed.Test_Type := 69, [18].VolumeTest.Detailed.element_data[0].Variable_code := 245, [18].VolumeTest.Detailed.element_data[0].prec_code := 2, [18].VolumeTest.Detailed.element_data[0].Unit_code := 165, [18].VolumeTest.Detailed.element_data[0].result_measurement := 214.21709, [18].VolumeTest.Detailed.element_data[1].Variable_code := 13, [18].VolumeTest.Detailed.element_data[1].prec_code := 3, [18].VolumeTest.Detailed.element_data[1].Unit_code := 12, [18].VolumeTest.Detailed.element_data[1].result_measurement := 1.5958865, [18].VolumeTest.Detailed.element_data[2].Variable_code := 247, [18].VolumeTest.Detailed.element_data[2].prec_code := 3, [18].VolumeTest.Detailed.element_data[2].Unit_code := 12, [18].VolumeTest.Detailed.element_data[2].result_measurement := 5.0145483, [18].VolumeTest.Detailed.element_data[3].Variable_code := 295, [18].VolumeTest.Detailed.element_data[3].prec_code := 3, [18].VolumeTest.Detailed.element_data[3].Unit_code := 12,
        [18].VolumeTest.Detailed.element_data[3].result_measurement := 5.0152373, [18].LeakTest.Detailed.element_data[0].result_measurement := -999.0, [19].Barcode := 'A252620388', [19].VolumeTest.UID := 25862, [19].VolumeTest.Basic.unique_id := 25862, [19].VolumeTest.Basic.channel_num := 1, [19].VolumeTest.Basic.program_num := 1, [19].VolumeTest.Basic.evaluation_code := 2, [19].VolumeTest.Basic.test_port := 1, [19].VolumeTest.Basic.year := 26, [19].VolumeTest.Basic.month := 6, [19].VolumeTest.Basic.date := 2, [19].VolumeTest.Basic.hour := 14, [19].VolumeTest.Basic.minute := 37, [19].VolumeTest.Basic.second := 42, [19].VolumeTest.Basic.flags := 12, [19].VolumeTest.Basic.Num_tests := 1, [19].VolumeTest.Basic.test_elements.test_type := 69, [19].VolumeTest.Basic.test_elements.test_eval := 2, [19].VolumeTest.Basic.test_elements.num_elements := 4, [19].VolumeTest.Detailed.unique_id := 25862, [19].VolumeTest.Detailed.num_elements := 4, [19].VolumeTest.Detailed.Test_Type := 69, [19].VolumeTest.Detailed.element_data[0].Variable_code := 245, [19].VolumeTest.Detailed.element_data[0].prec_code := 2, [19].VolumeTest.Detailed.element_data[0].Unit_code := 165, [19].VolumeTest.Detailed.element_data[0].result_measurement := 214.21709, [19].VolumeTest.Detailed.element_data[1].Variable_code := 13, [19].VolumeTest.Detailed.element_data[1].prec_code := 3, [19].VolumeTest.Detailed.element_data[1].Unit_code := 12, [19].VolumeTest.Detailed.element_data[1].result_measurement := 1.5958865, [19].VolumeTest.Detailed.element_data[2].Variable_code := 247, [19].VolumeTest.Detailed.element_data[2].prec_code := 3, [19].VolumeTest.Detailed.element_data[2].Unit_code := 12, [19].VolumeTest.Detailed.element_data[2].result_measurement := 5.0145483, [19].VolumeTest.Detailed.element_data[3].Variable_code := 295, [19].VolumeTest.Detailed.element_data[3].prec_code := 3, [19].VolumeTest.Detailed.element_data[3].Unit_code := 12, [19].VolumeTest.Detailed.element_data[3].result_measurement := 5.0152373, [19].LeakTest.Detailed.element_data[0].result_measurement := -999.0, [20].Barcode := 'A252620388', [20].VolumeTest.UID := 25862, [20].VolumeTest.Basic.unique_id := 25862, [20].VolumeTest.Basic.channel_num := 1, [20].VolumeTest.Basic.program_num := 1, [20].VolumeTest.Basic.evaluation_code := 2, [20].VolumeTest.Basic.test_port := 1, [20].VolumeTest.Basic.year := 26, [20].VolumeTest.Basic.month := 6, [20].VolumeTest.Basic.date := 2, [20].VolumeTest.Basic.hour := 14, [20].VolumeTest.Basic.minute := 37, [20].VolumeTest.Basic.second := 42, [20].VolumeTest.Basic.flags := 12, [20].VolumeTest.Basic.Num_tests := 1, [20].VolumeTest.Basic.test_elements.test_type := 69, [20].VolumeTest.Basic.test_elements.test_eval := 2, [20].VolumeTest.Basic.test_elements.num_elements := 4, [20].VolumeTest.Detailed.unique_id := 25862, [20].VolumeTest.Detailed.num_elements := 4,
        [20].VolumeTest.Detailed.Test_Type := 69, [20].VolumeTest.Detailed.element_data[0].Variable_code := 245, [20].VolumeTest.Detailed.element_data[0].prec_code := 2, [20].VolumeTest.Detailed.element_data[0].Unit_code := 165, [20].VolumeTest.Detailed.element_data[0].result_measurement := 214.21709, [20].VolumeTest.Detailed.element_data[1].Variable_code := 13, [20].VolumeTest.Detailed.element_data[1].prec_code := 3, [20].VolumeTest.Detailed.element_data[1].Unit_code := 12, [20].VolumeTest.Detailed.element_data[1].result_measurement := 1.5958865, [20].VolumeTest.Detailed.element_data[2].Variable_code := 247, [20].VolumeTest.Detailed.element_data[2].prec_code := 3, [20].VolumeTest.Detailed.element_data[2].Unit_code := 12, [20].VolumeTest.Detailed.element_data[2].result_measurement := 5.0145483, [20].VolumeTest.Detailed.element_data[3].Variable_code := 295, [20].VolumeTest.Detailed.element_data[3].prec_code := 3, [20].VolumeTest.Detailed.element_data[3].Unit_code := 12, [20].VolumeTest.Detailed.element_data[3].result_measurement := 5.0152373, [20].LeakTest.Detailed.element_data[0].result_measurement := -999.0, [21].Barcode := 'A252620388', [21].VolumeTest.UID := 25862, [21].VolumeTest.Basic.unique_id := 25862, [21].VolumeTest.Basic.channel_num := 1, [21].VolumeTest.Basic.program_num := 1, [21].VolumeTest.Basic.evaluation_code := 2, [21].VolumeTest.Basic.test_port := 1, [21].VolumeTest.Basic.year := 26, [21].VolumeTest.Basic.month := 6, [21].VolumeTest.Basic.date := 2, [21].VolumeTest.Basic.hour := 14, [21].VolumeTest.Basic.minute := 37, [21].VolumeTest.Basic.second := 42, [21].VolumeTest.Basic.flags := 12, [21].VolumeTest.Basic.Num_tests := 1, [21].VolumeTest.Basic.test_elements.test_type := 69, [21].VolumeTest.Basic.test_elements.test_eval := 2, [21].VolumeTest.Basic.test_elements.num_elements := 4, [21].VolumeTest.Detailed.unique_id := 25862, [21].VolumeTest.Detailed.num_elements := 4, [21].VolumeTest.Detailed.Test_Type := 69, [21].VolumeTest.Detailed.element_data[0].Variable_code := 245, [21].VolumeTest.Detailed.element_data[0].prec_code := 2, [21].VolumeTest.Detailed.element_data[0].Unit_code := 165, [21].VolumeTest.Detailed.element_data[0].result_measurement := 214.21709, [21].VolumeTest.Detailed.element_data[1].Variable_code := 13, [21].VolumeTest.Detailed.element_data[1].prec_code := 3, [21].VolumeTest.Detailed.element_data[1].Unit_code := 12, [21].VolumeTest.Detailed.element_data[1].result_measurement := 1.5958865, [21].VolumeTest.Detailed.element_data[2].Variable_code := 247, [21].VolumeTest.Detailed.element_data[2].prec_code := 3, [21].VolumeTest.Detailed.element_data[2].Unit_code := 12, [21].VolumeTest.Detailed.element_data[2].result_measurement := 5.0145483, [21].VolumeTest.Detailed.element_data[3].Variable_code := 295, [21].VolumeTest.Detailed.element_data[3].prec_code := 3, [21].VolumeTest.Detailed.element_data[3].Unit_code := 12, [21].VolumeTest.Detailed.element_data[3].result_measurement := 5.0152373, [21].LeakTest.Detailed.element_data[0].result_measurement := -999.0, [22].Barcode := 'A252620388', [22].VolumeTest.UID := 25862, [22].VolumeTest.Basic.unique_id := 25862, [22].VolumeTest.Basic.channel_num := 1,
        [22].VolumeTest.Basic.program_num := 1, [22].VolumeTest.Basic.evaluation_code := 2, [22].VolumeTest.Basic.test_port := 1, [22].VolumeTest.Basic.year := 26, [22].VolumeTest.Basic.month := 6, [22].VolumeTest.Basic.date := 2, [22].VolumeTest.Basic.hour := 14, [22].VolumeTest.Basic.minute := 37, [22].VolumeTest.Basic.second := 42, [22].VolumeTest.Basic.flags := 12, [22].VolumeTest.Basic.Num_tests := 1, [22].VolumeTest.Basic.test_elements.test_type := 69, [22].VolumeTest.Basic.test_elements.test_eval := 2, [22].VolumeTest.Basic.test_elements.num_elements := 4, [22].VolumeTest.Detailed.unique_id := 25862, [22].VolumeTest.Detailed.num_elements := 4, [22].VolumeTest.Detailed.Test_Type := 69, [22].VolumeTest.Detailed.element_data[0].Variable_code := 245, [22].VolumeTest.Detailed.element_data[0].prec_code := 2, [22].VolumeTest.Detailed.element_data[0].Unit_code := 165, [22].VolumeTest.Detailed.element_data[0].result_measurement := 214.21709, [22].VolumeTest.Detailed.element_data[1].Variable_code := 13, [22].VolumeTest.Detailed.element_data[1].prec_code := 3, [22].VolumeTest.Detailed.element_data[1].Unit_code := 12, [22].VolumeTest.Detailed.element_data[1].result_measurement := 1.5958865, [22].VolumeTest.Detailed.element_data[2].Variable_code := 247, [22].VolumeTest.Detailed.element_data[2].prec_code := 3, [22].VolumeTest.Detailed.element_data[2].Unit_code := 12, [22].VolumeTest.Detailed.element_data[2].result_measurement := 5.0145483, [22].VolumeTest.Detailed.element_data[3].Variable_code := 295, [22].VolumeTest.Detailed.element_data[3].prec_code := 3, [22].VolumeTest.Detailed.element_data[3].Unit_code := 12, [22].VolumeTest.Detailed.element_data[3].result_measurement := 5.0152373, [22].LeakTest.Detailed.element_data[0].result_measurement := -999.0, [23].Barcode := 'A252620388', [23].VolumeTest.UID := 25862, [23].VolumeTest.Basic.unique_id := 25862, [23].VolumeTest.Basic.channel_num := 1, [23].VolumeTest.Basic.program_num := 1, [23].VolumeTest.Basic.evaluation_code := 2, [23].VolumeTest.Basic.test_port := 1, [23].VolumeTest.Basic.year := 26, [23].VolumeTest.Basic.month := 6, [23].VolumeTest.Basic.date := 2, [23].VolumeTest.Basic.hour := 14, [23].VolumeTest.Basic.minute := 37, [23].VolumeTest.Basic.second := 42, [23].VolumeTest.Basic.flags := 12, [23].VolumeTest.Basic.Num_tests := 1, [23].VolumeTest.Basic.test_elements.test_type := 69, [23].VolumeTest.Basic.test_elements.test_eval := 2, [23].VolumeTest.Basic.test_elements.num_elements := 4, [23].VolumeTest.Detailed.unique_id := 25862, [23].VolumeTest.Detailed.num_elements := 4, [23].VolumeTest.Detailed.Test_Type := 69, [23].VolumeTest.Detailed.element_data[0].Variable_code := 245, [23].VolumeTest.Detailed.element_data[0].prec_code := 2, [23].VolumeTest.Detailed.element_data[0].Unit_code := 165, [23].VolumeTest.Detailed.element_data[0].result_measurement := 214.21709, [23].VolumeTest.Detailed.element_data[1].Variable_code := 13,
